LIN {X 0,Y 189.628,Z 761.034,A -85,B 0,C 180,E1 20728.512,E2 20728.512} C_VEL
LIN {X 0,Y 212.096,Z 753.744,A -85,B 0,C 180,E1 20739.808,E2 20739.808} C_VEL
LIN {X 0,Y 217.825,Z 751.684,A -85,B 0,C 180,E1 20741.718,E2 20741.718} C_VEL
LIN {X 0,Y 216.052,Z 752.751,A -85,B 0,C 180,E1 20742.834,E2 20742.834} C_VEL
LIN {X 0,Y 191.697,Z 765.754,A -85,B 0,C 180,E1 20753.818,E2 20753.818} C_VEL
LIN {X 0,Y 179.263,Z 772.931,A -85,B 0,C 180,E1 20765.112,E2 20765.112} C_VEL
LIN {X 0,Y 174.645,Z 775.618,A -85,B 0,C 180,E1 20774.979,E2 20774.979} C_VEL
LIN {X 0,Y 173.679,Z 775.979,A -85,B 0,C 180,E1 20785.018,E2 20785.018} C_VEL
LIN {X 0,Y 173.872,Z 777.551,A -85,B 0,C 180,E1 20790.002,E2 20790.002} C_VEL
LIN {X 0,Y 173.679,Z 777.533,A -85,B 0,C 180,E1 20794.986,E2 20794.986} C_VEL
LIN {X 0,Y 174.385,Z 774.615,A -85,B 0,C 180,E1 20802.496,E2 20802.496} C_VEL
LIN {X 0,Y 177.606,Z 765.224,A -85,B 0,C 180,E1 20812.481,E2 20812.481} C_VEL
LIN {X 0,Y 184.174,Z 750.072,A -85,B 0,C 180,E1 20821.354,E2 20821.354} C_VEL
LIN {X 0,Y 192.922,Z 729.385,A -85,B 0,C 180,E1 20828.739,E2 20828.739} C_VEL
LIN {X 0,Y 201.559,Z 704.57,A -85,B 0,C 180,E1 20834.347,E2 20834.347} C_VEL
LIN {X 0,Y 208.28,Z 677.85,A -85,B 0,C 180,E1 20838.151,E2 20838.151} C_VEL
LIN {X 0,Y 212.35,Z 649.044,A -85,B 0,C 180,E1 20840.62,E2 20840.62} C_VEL
LIN {X 0,Y 213.87,Z 640.631,A -85,B 0,C 180,E1 20841.448,E2 20841.448} C_VEL
LIN {X 0,Y 203.795,Z 603.79,A -85,B 0,C 180,E1 20848.943,E2 20848.943} C_VEL
LIN {X 0,Y 198.917,Z 565.383,A -85,B 0,C 180,E1 20858.768,E2 20858.768} C_VEL
LIN {X 0,Y 197.323,Z 560.632,A -85,B 0,C 180,E1 20863.341,E2 20863.341} C_VEL
LIN {X 0,Y 198.795,Z 561.143,A -85,B 0,C 180,E1 20875.653,E2 20875.653} C_VEL
LIN {X 0,Y 203.113,Z 569.312,A -85,B 0,C 180,E1 20882.168,E2 20882.168} C_VEL
LIN {X 0,Y 209.323,Z 580.62,A -85,B 0,C 180,E1 20887.904,E2 20887.904} C_VEL
LIN {X 0,Y 217.509,Z 597.767,A -85,B 0,C 180,E1 20893.44,E2 20893.44} C_VEL
LIN {X 0,Y 225.175,Z 619.284,A -85,B 0,C 180,E1 20897.758,E2 20897.758} C_VEL
LIN {X 0,Y 226.031,Z 622.404,A -85,B 0,C 180,E1 20898.235,E2 20898.235} C_VEL
LIN {X 0,Y 222.435,Z 652.717,A -85,B 0,C 180,E1 20899.64,E2 20899.64} C_VEL
LIN {X 0,Y 219.352,Z 667.346,A -85,B 0,C 180,E1 20900.828,E2 20900.828} C_VEL
LIN {X 0,Y 212.303,Z 683.08,A -85,B 0,C 180,E1 20901.722,E2 20901.722} C_VEL
LIN {X 0,Y 205.16,Z 696.073,A -85,B 0,C 180,E1 20902.814,E2 20902.814} C_VEL
LIN {X 0,Y 204.418,Z 697.811,A -85,B 0,C 180,E1 20903.1,E2 20903.1} C_VEL
LIN {X 0,Y 194.005,Z 720.009,A -85,B 0,C 180,E1 20907.989,E2 20907.989} C_VEL
LIN {X 0,Y 183.31,Z 738.179,A -85,B 0,C 180,E1 20914.591,E2 20914.591} C_VEL
LIN {X 0,Y 174.062,Z 751.886,A -85,B 0,C 180,E1 20923.249,E2 20923.249} C_VEL
LIN {X 0,Y 169.021,Z 758.609,A -85,B 0,C 180,E1 20931.319,E2 20931.319} C_VEL
LIN {X 0,Y 166.585,Z 760.947,A -85,B 0,C 180,E1 20937.075,E2 20937.075} C_VEL
LIN {X 0,Y 165.326,Z 760.854,A -85,B 0,C 180,E1 20945.902,E2 20945.902} C_VEL
LIN {X 0,Y 167.356,Z 755.765,A -85,B 0,C 180,E1 20955.642,E2 20955.642} C_VEL
LIN {X 0,Y 171.894,Z 745.002,A -85,B 0,C 180,E1 20964.962,E2 20964.962} C_VEL
LIN {X 0,Y 178.888,Z 728.891,A -85,B 0,C 180,E1 20973.02,E2 20973.02} C_VEL
LIN {X 0,Y 187.361,Z 707.541,A -85,B 0,C 180,E1 20979.56,E2 20979.56} C_VEL
LIN {X 0,Y 195.39,Z 682.576,A -85,B 0,C 180,E1 20984.249,E2 20984.249} C_VEL
LIN {X 0,Y 201.6,Z 654.272,A -85,B 0,C 180,E1 20987.42,E2 20987.42} C_VEL
LIN {X 0,Y 205.022,Z 624.843,A -85,B 0,C 180,E1 20989.044,E2 20989.044} C_VEL
LIN {X 0,Y 204.978,Z 613.442,A -85,B 0,C 180,E1 20989.593,E2 20989.593} C_VEL
LIN {X 0,Y 193.143,Z 583.54,A -85,B 0,C 180,E1 20994.123,E2 20994.123} C_VEL
LIN {X 0,Y 184.516,Z 566.701,A -85,B 0,C 180,E1 20997.701,E2 20997.701} C_VEL
LIN {X 0,Y 180.361,Z 568.066,A -85,B 0,C 180,E1 20999.224,E2 20999.224} C_VEL
LIN {X 0,Y 192.479,Z 600.451,A -85,B 0,C 180,E1 21006.012,E2 21006.012} C_VEL
LIN {X 0,Y 201.469,Z 633.152,A -85,B 0,C 180,E1 21012.744,E2 21012.744} C_VEL
LIN {X 0,Y 192.439,Z 663.924,A -85,B 0,C 180,E1 21017.77,E2 21017.77} C_VEL
LIN {X 0,Y 181.952,Z 694.148,A -85,B 0,C 180,E1 21024.976,E2 21024.976} C_VEL
LIN {X 0,Y 173.22,Z 719.714,A -85,B 0,C 180,E1 21034.171,E2 21034.171} C_VEL
LIN {X 0,Y 167.935,Z 738.514,A -85,B 0,C 180,E1 21044.355,E2 21044.355} C_VEL
LIN {X 0,Y 166.031,Z 751.24,A -85,B 0,C 180,E1 21054.779,E2 21054.779} C_VEL
LIN {X 0,Y 166.344,Z 758.967,A -85,B 0,C 180,E1 21065.198,E2 21065.198} C_VEL
LIN {X 0,Y 169.63,Z 762.701,A -85,B 0,C 180,E1 21075.471,E2 21075.471} C_VEL
LIN {X 0,Y 182.8,Z 762.307,A -85,B 0,C 180,E1 21089.681,E2 21089.681} C_VEL
LIN {X 0,Y 207.708,Z 755.77,A -85,B 0,C 180,E1 21101.58,E2 21101.58} C_VEL
LIN {X 0,Y 207.442,Z 756.059,A -85,B 0,C 180,E1 21102.411,E2 21102.411} C_VEL
LIN {X 0,Y 182.073,Z 767.938,A -85,B 0,C 180,E1 21114.541,E2 21114.541} C_VEL
LIN {X 0,Y 168.849,Z 774.269,A -85,B 0,C 180,E1 21129.057,E2 21129.057} C_VEL
LIN {X 0,Y 165.827,Z 774.847,A -85,B 0,C 180,E1 21143.471,E2 21143.471} C_VEL
LIN {X 0,Y 165.967,Z 777.14,A -85,B 0,C 180,E1 21150.134,E2 21150.134} C_VEL
LIN {X 0,Y 165.798,Z 777.161,A -85,B 0,C 180,E1 21155.224,E2 21155.224} C_VEL
LIN {X 0,Y 166.57,Z 774.369,A -85,B 0,C 180,E1 21163.092,E2 21163.092} C_VEL
LIN {X 0,Y 170.156,Z 765.137,A -85,B 0,C 180,E1 21173.523,E2 21173.523} C_VEL
LIN {X 0,Y 177.467,Z 749.999,A -85,B 0,C 180,E1 21182.827,E2 21182.827} C_VEL
LIN {X 0,Y 186.742,Z 729.883,A -85,B 0,C 180,E1 21190.277,E2 21190.277} C_VEL
LIN {X 0,Y 195.714,Z 706.541,A -85,B 0,C 180,E1 21195.771,E2 21195.771} C_VEL
LIN {X 0,Y 203.105,Z 680.501,A -85,B 0,C 180,E1 21199.69,E2 21199.69} C_VEL
LIN {X 0,Y 207.927,Z 651.201,A -85,B 0,C 180,E1 21202.351,E2 21202.351} C_VEL
LIN {X 0,Y 208.329,Z 642.972,A -85,B 0,C 180,E1 21202.993,E2 21202.993} C_VEL
LIN {X 0,Y 198.886,Z 594.701,A -85,B 0,C 180,E1 21213.925,E2 21213.925} C_VEL
LIN {X 0,Y 197.153,Z 572.184,A -85,B 0,C 180,E1 21220.11,E2 21220.11} C_VEL
LIN {X 0,Y 196.152,Z 568.38,A -85,B 0,C 180,E1 21223.777,E2 21223.777} C_VEL
LIN {X 0,Y 197.478,Z 568.897,A -85,B 0,C 180,E1 21235.212,E2 21235.212} C_VEL
LIN {X 0,Y 201.518,Z 576.988,A -85,B 0,C 180,E1 21241.702,E2 21241.702} C_VEL
LIN {X 0,Y 208.238,Z 589.979,A -85,B 0,C 180,E1 21248.076,E2 21248.076} C_VEL
LIN {X 0,Y 216.187,Z 608.855,A -85,B 0,C 180,E1 21253.614,E2 21253.614} C_VEL
LIN {X 0,Y 221.286,Z 624.924,A -85,B 0,C 180,E1 21256.677,E2 21256.677} C_VEL
LIN {X 0,Y 217.341,Z 654.833,A -85,B 0,C 180,E1 21258.13,E2 21258.13} C_VEL
LIN {X 0,Y 209.921,Z 682.887,A -85,B 0,C 180,E1 21260.85,E2 21260.85} C_VEL
LIN {X 0,Y 204.418,Z 697.811,A -85,B 0,C 180,E1 21263.1,E2 21263.1} C_VEL
LIN {X 0,Y 195.677,Z 711.55,A -85,B 0,C 180,E1 21264.989,E2 21264.989} C_VEL
LIN {X 0,Y 187.156,Z 722.49,A -85,B 0,C 180,E1 21266.974,E2 21266.974} C_VEL
LIN {X 0,Y 186.262,Z 723.922,A -85,B 0,C 180,E1 21267.391,E2 21267.391} C_VEL
LIN {X 0,Y 175.216,Z 741.093,A -85,B 0,C 180,E1 21274.304,E2 21274.304} C_VEL
LIN {X 0,Y 165.895,Z 753.645,A -85,B 0,C 180,E1 21283.304,E2 21283.304} C_VEL
LIN {X 0,Y 160.55,Z 759.928,A -85,B 0,C 180,E1 21292.228,E2 21292.228} C_VEL
LIN {X 0,Y 157.683,Z 761.83,A -85,B 0,C 180,E1 21301.411,E2 21301.411} C_VEL
LIN {X 0,Y 158.41,Z 758.563,A -85,B 0,C 180,E1 21312.308,E2 21312.308} C_VEL
LIN {X 0,Y 162.077,Z 750.222,A -85,B 0,C 180,E1 21321.994,E2 21321.994} C_VEL
LIN {X 0,Y 168.815,Z 735.543,A -85,B 0,C 180,E1 21331.278,E2 21331.278} C_VEL
LIN {X 0,Y 177.046,Z 716.518,A -85,B 0,C 180,E1 21338.463,E2 21338.463} C_VEL
LIN {X 0,Y 186.063,Z 692.234,A -85,B 0,C 180,E1 21344.08,E2 21344.08} C_VEL
LIN {X 0,Y 193.442,Z 664.259,A -85,B 0,C 180,E1 21347.933,E2 21347.933} C_VEL
LIN {X 0,Y 198.021,Z 636.087,A -85,B 0,C 180,E1 21350.011,E2 21350.011} C_VEL
LIN {X 0,Y 198.961,Z 616.022,A -85,B 0,C 180,E1 21350.912,E2 21350.912} C_VEL
LIN {X 0,Y 187.164,Z 586.134,A -85,B 0,C 180,E1 21355.733,E2 21355.733} C_VEL
LIN {X 0,Y 181.93,Z 576.305,A -85,B 0,C 180,E1 21357.983,E2 21357.983} C_VEL
LIN {X 0,Y 177.718,Z 578.756,A -85,B 0,C 180,E1 21359.29,E2 21359.29} C_VEL
LIN {X 0,Y 177.042,Z 578.811,A -85,B 0,C 180,E1 21359.673,E2 21359.673} C_VEL
LIN {X 0,Y 187.669,Z 609.878,A -85,B 0,C 180,E1 21366.47,E2 21366.47} C_VEL
LIN {X 0,Y 194.332,Z 635.863,A -85,B 0,C 180,E1 21372.116,E2 21372.116} C_VEL
LIN {X 0,Y 182.885,Z 670.726,A -85,B 0,C 180,E1 21378.229,E2 21378.229} C_VEL
LIN {X 0,Y 172.181,Z 700.201,A -85,B 0,C 180,E1 21386.166,E2 21386.166} C_VEL
LIN {X 0,Y 164.136,Z 723.35,A -85,B 0,C 180,E1 21395.557,E2 21395.557} C_VEL
LIN {X 0,Y 159.49,Z 741.202,A -85,B 0,C 180,E1 21406.311,E2 21406.311} C_VEL
LIN {X 0,Y 157.983,Z 753.046,A -85,B 0,C 180,E1 21417.255,E2 21417.255} C_VEL
LIN {X 0,Y 158.965,Z 760.202,A -85,B 0,C 180,E1 21428.179,E2 21428.179} C_VEL
LIN {X 0,Y 165.439,Z 763.919,A -85,B 0,C 180,E1 21441.39,E2 21441.39} C_VEL
LIN {X 0,Y 183.212,Z 762.391,A -85,B 0,C 180,E1 21455.2,E2 21455.2} C_VEL
LIN {X 0,Y 197.664,Z 759.231,A -85,B 0,C 180,E1 21461.464,E2 21461.464} C_VEL
LIN {X 0,Y 197.434,Z 759.516,A -85,B 0,C 180,E1 21462.426,E2 21462.426} C_VEL
LIN {X 0,Y 172.433,Z 769.611,A -85,B 0,C 180,E1 21475.334,E2 21475.334} C_VEL
LIN {X 0,Y 160.311,Z 774.163,A -85,B 0,C 180,E1 21490.246,E2 21490.246} C_VEL
LIN {X 0,Y 157.942,Z 774.318,A -85,B 0,C 180,E1 21503.143,E2 21503.143} C_VEL
LIN {X 0,Y 158.103,Z 776.683,A -85,B 0,C 180,E1 21510.002,E2 21510.002} C_VEL
LIN {X 0,Y 157.889,Z 776.788,A -85,B 0,C 180,E1 21515.487,E2 21515.487} C_VEL
LIN {X 0,Y 158.753,Z 774.123,A -85,B 0,C 180,E1 21523.749,E2 21523.749} C_VEL
LIN {X 0,Y 162.797,Z 765.073,A -85,B 0,C 180,E1 21534.655,E2 21534.655} C_VEL
LIN {X 0,Y 170.744,Z 750.181,A -85,B 0,C 180,E1 21544.294,E2 21544.294} C_VEL
LIN {X 0,Y 180.725,Z 730.409,A -85,B 0,C 180,E1 21551.914,E2 21551.914} C_VEL
LIN {X 0,Y 190.329,Z 707.567,A -85,B 0,C 180,E1 21557.463,E2 21557.463} C_VEL
LIN {X 0,Y 198.596,Z 680.998,A -85,B 0,C 180,E1 21561.549,E2 21561.549} C_VEL
LIN {X 0,Y 203.976,Z 651.61,A -85,B 0,C 180,E1 21564.25,E2 21564.25} C_VEL
LIN {X 0,Y 204.189,Z 645.575,A -85,B 0,C 180,E1 21564.854,E2 21564.854} C_VEL
LIN {X 0,Y 196.541,Z 598.917,A -85,B 0,C 180,E1 21575.806,E2 21575.806} C_VEL
LIN {X 0,Y 195.582,Z 579.18,A -85,B 0,C 180,E1 21581.253,E2 21581.253} C_VEL
LIN {X 0,Y 194.934,Z 576.15,A -85,B 0,C 180,E1 21584.453,E2 21584.453} C_VEL
LIN {X 0,Y 196.294,Z 576.937,A -85,B 0,C 180,E1 21595.054,E2 21595.054} C_VEL
LIN {X 0,Y 200.005,Z 584.838,A -85,B 0,C 180,E1 21601.317,E2 21601.317} C_VEL
LIN {X 0,Y 205.971,Z 597.331,A -85,B 0,C 180,E1 21607.35,E2 21607.35} C_VEL
LIN {X 0,Y 212.922,Z 614.88,A -85,B 0,C 180,E1 21612.541,E2 21612.541} C_VEL
LIN {X 0,Y 216.636,Z 628.564,A -85,B 0,C 180,E1 21615.096,E2 21615.096} C_VEL
LIN {X 0,Y 212.183,Z 658.001,A -85,B 0,C 180,E1 21616.625,E2 21616.625} C_VEL
LIN {X 0,Y 204.222,Z 685.488,A -85,B 0,C 180,E1 21619.428,E2 21619.428} C_VEL
LIN {X 0,Y 194.017,Z 709.671,A -85,B 0,C 180,E1 21623.652,E2 21623.652} C_VEL
LIN {X 0,Y 186.262,Z 723.922,A -85,B 0,C 180,E1 21627.391,E2 21627.391} C_VEL
LIN {X 0,Y 176.493,Z 734.878,A -85,B 0,C 180,E1 21630.447,E2 21630.447} C_VEL
LIN {X 0,Y 167.686,Z 743.126,A -85,B 0,C 180,E1 21633.613,E2 21633.613} C_VEL
LIN {X 0,Y 166.844,Z 744.164,A -85,B 0,C 180,E1 21634.201,E2 21634.201} C_VEL
LIN {X 0,Y 157.571,Z 755.542,A -85,B 0,C 180,E1 21643.595,E2 21643.595} C_VEL
LIN {X 0,Y 152.001,Z 761.137,A -85,B 0,C 180,E1 21653.438,E2 21653.438} C_VEL
LIN {X 0,Y 150.056,Z 762.194,A -85,B 0,C 180,E1 21659.811,E2 21659.811} C_VEL
LIN {X 0,Y 149.873,Z 760.404,A -85,B 0,C 180,E1 21669.363,E2 21669.363} C_VEL
LIN {X 0,Y 153.178,Z 753.143,A -85,B 0,C 180,E1 21680.145,E2 21680.145} C_VEL
LIN {X 0,Y 159.38,Z 740.172,A -85,B 0,C 180,E1 21689.998,E2 21689.998} C_VEL
LIN {X 0,Y 167.983,Z 721.865,A -85,B 0,C 180,E1 21698.084,E2 21698.084} C_VEL
LIN {X 0,Y 177.152,Z 699.254,A -85,B 0,C 180,E1 21704.173,E2 21704.173} C_VEL
LIN {X 0,Y 185.408,Z 672.3,A -85,B 0,C 180,E1 21708.529,E2 21708.529} C_VEL
LIN {X 0,Y 191.102,Z 643.534,A -85,B 0,C 180,E1 21711.104,E2 21711.104} C_VEL
LIN {X 0,Y 192.851,Z 618.067,A -85,B 0,C 180,E1 21712.373,E2 21712.373} C_VEL
LIN {X 0,Y 181.472,Z 589.025,A -85,B 0,C 180,E1 21717.367,E2 21717.367} C_VEL
LIN {X 0,Y 179.739,Z 586.175,A -85,B 0,C 180,E1 21718.124,E2 21718.124} C_VEL
LIN {X 0,Y 175.253,Z 589.51,A -85,B 0,C 180,E1 21719.489,E2 21719.489} C_VEL
LIN {X 0,Y 173.535,Z 589.694,A -85,B 0,C 180,E1 21720.289,E2 21720.289} C_VEL
LIN {X 0,Y 182.849,Z 620.052,A -85,B 0,C 180,E1 21727.243,E2 21727.243} C_VEL
LIN {X 0,Y 186.67,Z 638.028,A -85,B 0,C 180,E1 21731.303,E2 21731.303} C_VEL
LIN {X 0,Y 174.947,Z 672.291,A -85,B 0,C 180,E1 21737.626,E2 21737.626} C_VEL
LIN {X 0,Y 164.226,Z 701.045,A -85,B 0,C 180,E1 21745.784,E2 21745.784} C_VEL
LIN {X 0,Y 155.999,Z 724.212,A -85,B 0,C 180,E1 21755.718,E2 21755.718} C_VEL
LIN {X 0,Y 151.395,Z 741.872,A -85,B 0,C 180,E1 21767.033,E2 21767.033} C_VEL
LIN {X 0,Y 150.106,Z 753.609,A -85,B 0,C 180,E1 21778.552,E2 21778.552} C_VEL
LIN {X 0,Y 151.972,Z 761.332,A -85,B 0,C 180,E1 21791.447,E2 21791.447} C_VEL
LIN {X 0,Y 163.147,Z 764.871,A -85,B 0,C 180,E1 21807.538,E2 21807.538} C_VEL
LIN {X 0,Y 188.299,Z 761.982,A -85,B 0,C 180,E1 21821.617,E2 21821.617} C_VEL
LIN {X 0,Y 176.931,Z 765.985,A -85,B 0,C 180,E1 21826.98,E2 21826.98} C_VEL
LIN {X 0,Y 157.636,Z 772.371,A -85,B 0,C 180,E1 21841.407,E2 21841.407} C_VEL
LIN {X 0,Y 150.423,Z 773.203,A -85,B 0,C 180,E1 21858.429,E2 21858.429} C_VEL
LIN {X 0,Y 150.174,Z 772.989,A -85,B 0,C 180,E1 21861.334,E2 21861.334} C_VEL
LIN {X 0,Y 150.225,Z 776.245,A -85,B 0,C 180,E1 21870.002,E2 21870.002} C_VEL
LIN {X 0,Y 149.986,Z 776.416,A -85,B 0,C 180,E1 21875.777,E2 21875.777} C_VEL
LIN {X 0,Y 150.972,Z 773.862,A -85,B 0,C 180,E1 21884.473,E2 21884.473} C_VEL
LIN {X 0,Y 155.506,Z 765.02,A -85,B 0,C 180,E1 21895.894,E2 21895.894} C_VEL
LIN {X 0,Y 164.155,Z 750.364,A -85,B 0,C 180,E1 21905.878,E2 21905.878} C_VEL
LIN {X 0,Y 174.871,Z 731.01,A -85,B 0,C 180,E1 21913.66,E2 21913.66} C_VEL
LIN {X 0,Y 185.907,Z 706.743,A -85,B 0,C 180,E1 21919.615,E2 21919.615} C_VEL
LIN {X 0,Y 194.859,Z 679.634,A -85,B 0,C 180,E1 21923.714,E2 21923.714} C_VEL
LIN {X 0,Y 200.409,Z 649.217,A -85,B 0,C 180,E1 21926.563,E2 21926.563} C_VEL
LIN {X 0,Y 194.426,Z 602.064,A -85,B 0,C 180,E1 21937.983,E2 21937.983} C_VEL
LIN {X 0,Y 194.16,Z 586.04,A -85,B 0,C 180,E1 21942.507,E2 21942.507} C_VEL
LIN {X 0,Y 193.742,Z 583.92,A -85,B 0,C 180,E1 21945.136,E2 21945.136} C_VEL
LIN {X 0,Y 195.011,Z 584.643,A -85,B 0,C 180,E1 21954.595,E2 21954.595} C_VEL
LIN {X 0,Y 198.777,Z 593.064,A -85,B 0,C 180,E1 21961.236,E2 21961.236} C_VEL
LIN {X 0,Y 204.715,Z 606.886,A -85,B 0,C 180,E1 21967.435,E2 21967.435} C_VEL
LIN {X 0,Y 211.136,Z 625.779,A -85,B 0,C 180,E1 21972.483,E2 21972.483} C_VEL
LIN {X 0,Y 212.219,Z 630.971,A -85,B 0,C 180,E1 21973.385,E2 21973.385} C_VEL
LIN {X 0,Y 207.312,Z 660.175,A -85,B 0,C 180,E1 21974.974,E2 21974.974} C_VEL
LIN {X 0,Y 198.833,Z 687.616,A -85,B 0,C 180,E1 21977.863,E2 21977.863} C_VEL
LIN {X 0,Y 187.723,Z 712.088,A -85,B 0,C 180,E1 21982.312,E2 21982.312} C_VEL
LIN {X 0,Y 175.442,Z 732.306,A -85,B 0,C 180,E1 21988.436,E2 21988.436} C_VEL
LIN {X 0,Y 166.844,Z 744.164,A -85,B 0,C 180,E1 21994.201,E2 21994.201} C_VEL
LIN {X 0,Y 157.636,Z 751.717,A -85,B 0,C 180,E1 21998.746,E2 21998.746} C_VEL
LIN {X 0,Y 149.113,Z 757.363,A -85,B 0,C 180,E1 22004.075,E2 22004.075} C_VEL
LIN {X 0,Y 144.969,Z 761.155,A -85,B 0,C 180,E1 22011.348,E2 22011.348} C_VEL
LIN {X 0,Y 142.516,Z 762.55,A -85,B 0,C 180,E1 22018.031,E2 22018.031} C_VEL
LIN {X 0,Y 141.776,Z 761.214,A -85,B 0,C 180,E1 22028.126,E2 22028.126} C_VEL
LIN {X 0,Y 145.085,Z 754.21,A -85,B 0,C 180,E1 22039.906,E2 22039.906} C_VEL
LIN {X 0,Y 151.179,Z 742.096,A -85,B 0,C 180,E1 22049.998,E2 22049.998} C_VEL
LIN {X 0,Y 159.434,Z 725.534,A -85,B 0,C 180,E1 22058.158,E2 22058.158} C_VEL
LIN {X 0,Y 169.28,Z 703.118,A -85,B 0,C 180,E1 22064.847,E2 22064.847} C_VEL
LIN {X 0,Y 178.381,Z 676.175,A -85,B 0,C 180,E1 22069.598,E2 22069.598} C_VEL
LIN {X 0,Y 184.523,Z 647.904,A -85,B 0,C 180,E1 22072.416,E2 22072.416} C_VEL
LIN {X 0,Y 187.067,Z 620.816,A -85,B 0,C 180,E1 22073.825,E2 22073.825} C_VEL
LIN {X 0,Y 177.841,Z 596.291,A -85,B 0,C 180,E1 22078.147,E2 22078.147} C_VEL
LIN {X 0,Y 170.407,Z 600.502,A -85,B 0,C 180,E1 22080.569,E2 22080.569} C_VEL
LIN {X 0,Y 169.696,Z 600.579,A -85,B 0,C 180,E1 22081.052,E2 22081.052} C_VEL
LIN {X 0,Y 178.051,Z 631.757,A -85,B 0,C 180,E1 22088.546,E2 22088.546} C_VEL
LIN {X 0,Y 179.24,Z 639.536,A -85,B 0,C 180,E1 22090.354,E2 22090.354} C_VEL
LIN {X 0,Y 167.255,Z 673.247,A -85,B 0,C 180,E1 22096.86,E2 22096.86} C_VEL
LIN {X 0,Y 156.233,Z 701.911,A -85,B 0,C 180,E1 22105.419,E2 22105.419} C_VEL
LIN {X 0,Y 147.833,Z 724.983,A -85,B 0,C 180,E1 22115.894,E2 22115.894} C_VEL
LIN {X 0,Y 143.328,Z 742.475,A -85,B 0,C 180,E1 22127.836,E2 22127.836} C_VEL
LIN {X 0,Y 142.307,Z 754.116,A -85,B 0,C 180,E1 22139.992,E2 22139.992} C_VEL
LIN {X 0,Y 144.21,Z 761.258,A -85,B 0,C 180,E1 22152.072,E2 22152.072} C_VEL
LIN {X 0,Y 156.198,Z 765.58,A -85,B 0,C 180,E1 22168.875,E2 22168.875} C_VEL
LIN {X 0,Y 178.13,Z 764.364,A -85,B 0,C 180,E1 22181.495,E2 22181.495} C_VEL
LIN {X 0,Y 176.293,Z 765.001,A -85,B 0,C 180,E1 22182.838,E2 22182.838} C_VEL
LIN {X 0,Y 150.624,Z 771.993,A -85,B 0,C 180,E1 22199.942,E2 22199.942} C_VEL
LIN {X 0,Y 142.646,Z 772.227,A -85,B 0,C 180,E1 22217.788,E2 22217.788} C_VEL
LIN {X 0,Y 142.349,Z 772.425,A -85,B 0,C 180,E1 22220.853,E2 22220.853} C_VEL
LIN {X 0,Y 142.32,Z 775.803,A -85,B 0,C 180,E1 22230.003,E2 22230.003} C_VEL
LIN {X 0,Y 142.078,Z 776.044,A -85,B 0,C 180,E1 22236.099,E2 22236.099} C_VEL
LIN {X 0,Y 143.207,Z 773.601,A -85,B 0,C 180,E1 22245.276,E2 22245.276} C_VEL
LIN {X 0,Y 148.304,Z 764.995,A -85,B 0,C 180,E1 22257.253,E2 22257.253} C_VEL
LIN {X 0,Y 157.692,Z 750.587,A -85,B 0,C 180,E1 22267.595,E2 22267.595} C_VEL
LIN {X 0,Y 169.211,Z 731.612,A -85,B 0,C 180,E1 22275.517,E2 22275.517} C_VEL
LIN {X 0,Y 180.478,Z 708.981,A -85,B 0,C 180,E1 22281.286,E2 22281.286} C_VEL
LIN {X 0,Y 189.959,Z 683.295,A -85,B 0,C 180,E1 22285.385,E2 22285.385} C_VEL
LIN {X 0,Y 196.796,Z 652.858,A -85,B 0,C 180,E1 22288.331,E2 22288.331} C_VEL
LIN {X 0,Y 192.592,Z 604.507,A -85,B 0,C 180,E1 22300.384,E2 22300.384} C_VEL
LIN {X 0,Y 192.834,Z 592.695,A -85,B 0,C 180,E1 22303.915,E2 22303.915} C_VEL
LIN {X 0,Y 192.853,Z 591.48,A -85,B 0,C 180,E1 22311.003,E2 22311.003} C_VEL
LIN {X 0,Y 193.939,Z 592.919,A -85,B 0,C 180,E1 22314.705,E2 22314.705} C_VEL
LIN {X 0,Y 197.491,Z 601.298,A -85,B 0,C 180,E1 22321.089,E2 22321.089} C_VEL
LIN {X 0,Y 203.135,Z 615.947,A -85,B 0,C 180,E1 22327.259,E2 22327.259} C_VEL
LIN {X 0,Y 208.085,Z 632.68,A -85,B 0,C 180,E1 22331.523,E2 22331.523} C_VEL
LIN {X 0,Y 202.816,Z 662.049,A -85,B 0,C 180,E1 22333.209,E2 22333.209} C_VEL
LIN {X 0,Y 193.83,Z 689.253,A -85,B 0,C 180,E1 22336.144,E2 22336.144} C_VEL
LIN {X 0,Y 181.769,Z 714.063,A -85,B 0,C 180,E1 22340.802,E2 22340.802} C_VEL
LIN {X 0,Y 169.187,Z 733.463,A -85,B 0,C 180,E1 22346.882,E2 22346.882} C_VEL
LIN {X 0,Y 157.189,Z 748.569,A -85,B 0,C 180,E1 22355.178,E2 22355.178} C_VEL
LIN {X 0,Y 149.113,Z 757.363,A -85,B 0,C 180,E1 22364.075,E2 22364.075} C_VEL
LIN {X 0,Y 143.739,Z 760.436,A -85,B 0,C 180,E1 22368.613,E2 22368.613} C_VEL
LIN {X 0,Y 135.213,Z 762.818,A -85,B 0,C 180,E1 22375.929,E2 22375.929} C_VEL
LIN {X 0,Y 134.834,Z 762.825,A -85,B 0,C 180,E1 22376.85,E2 22376.85} C_VEL
LIN {X 0,Y 133.728,Z 762.462,A -85,B 0,C 180,E1 22384.537,E2 22384.537} C_VEL
LIN {X 0,Y 136.034,Z 757.056,A -85,B 0,C 180,E1 22397.179,E2 22397.179} C_VEL
LIN {X 0,Y 141.786,Z 746.054,A -85,B 0,C 180,E1 22408.473,E2 22408.473} C_VEL
LIN {X 0,Y 150.438,Z 729.936,A -85,B 0,C 180,E1 22417.8,E2 22417.8} C_VEL
LIN {X 0,Y 160.484,Z 709.031,A -85,B 0,C 180,E1 22424.983,E2 22424.983} C_VEL
LIN {X 0,Y 170.049,Z 683.806,A -85,B 0,C 180,E1 22430.157,E2 22430.157} C_VEL
LIN {X 0,Y 177.316,Z 655.689,A -85,B 0,C 180,E1 22433.502,E2 22433.502} C_VEL
LIN {X 0,Y 181.379,Z 625.224,A -85,B 0,C 180,E1 22435.256,E2 22435.256} C_VEL
LIN {X 0,Y 175.984,Z 607.958,A -85,B 0,C 180,E1 22438.058,E2 22438.058} C_VEL
LIN {X 0,Y 170.976,Z 608.808,A -85,B 0,C 180,E1 22439.793,E2 22439.793} C_VEL
LIN {X 0,Y 167.395,Z 611.489,A -85,B 0,C 180,E1 22440.985,E2 22440.985} C_VEL
LIN {X 0,Y 165.424,Z 611.345,A -85,B 0,C 180,E1 22441.922,E2 22441.922} C_VEL
LIN {X 0,Y 172.131,Z 640.155,A -85,B 0,C 180,E1 22449.214,E2 22449.214} C_VEL
LIN {X 0,Y 159.427,Z 674.544,A -85,B 0,C 180,E1 22456.147,E2 22456.147} C_VEL
LIN {X 0,Y 148.134,Z 702.785,A -85,B 0,C 180,E1 22465.055,E2 22465.055} C_VEL
LIN {X 0,Y 139.363,Z 726.814,A -85,B 0,C 180,E1 22476.765,E2 22476.765} C_VEL
LIN {X 0,Y 135.1,Z 744.15,A -85,B 0,C 180,E1 22489.802,E2 22489.802} C_VEL
LIN {X 0,Y 134.573,Z 755.654,A -85,B 0,C 180,E1 22503.205,E2 22503.205} C_VEL
LIN {X 0,Y 139.305,Z 763.478,A -85,B 0,C 180,E1 22518.955,E2 22518.955} C_VEL
LIN {X 0,Y 156.335,Z 766.521,A -85,B 0,C 180,E1 22535.38,E2 22535.38} C_VEL
LIN {X 0,Y 167.045,Z 766.219,A -85,B 0,C 180,E1 22540.963,E2 22540.963} C_VEL
LIN {X 0,Y 167.99,Z 766.334,A -85,B 0,C 180,E1 22542.149,E2 22542.149} C_VEL
LIN {X 0,Y 143.704,Z 771.569,A -85,B 0,C 180,E1 22558.333,E2 22558.333} C_VEL
LIN {X 0,Y 134.828,Z 770.937,A -85,B 0,C 180,E1 22577.889,E2 22577.889} C_VEL
LIN {X 0,Y 134.421,Z 775.359,A -85,B 0,C 180,E1 22590.003,E2 22590.003} C_VEL
LIN {X 0,Y 134.178,Z 775.674,A -85,B 0,C 180,E1 22596.46,E2 22596.46} C_VEL
LIN {X 0,Y 135.492,Z 773.351,A -85,B 0,C 180,E1 22606.169,E2 22606.169} C_VEL
LIN {X 0,Y 141.208,Z 764.976,A -85,B 0,C 180,E1 22618.746,E2 22618.746} C_VEL
LIN {X 0,Y 151.396,Z 750.83,A -85,B 0,C 180,E1 22629.453,E2 22629.453} C_VEL
LIN {X 0,Y 163.734,Z 732.201,A -85,B 0,C 180,E1 22637.504,E2 22637.504} C_VEL
LIN {X 0,Y 176.392,Z 708.649,A -85,B 0,C 180,E1 22643.593,E2 22643.593} C_VEL
LIN {X 0,Y 187.2,Z 680.965,A -85,B 0,C 180,E1 22647.857,E2 22647.857} C_VEL
LIN {X 0,Y 193.234,Z 655.109,A -85,B 0,C 180,E1 22650.483,E2 22650.483} C_VEL
LIN {X 0,Y 191.241,Z 606.707,A -85,B 0,C 180,E1 22662.883,E2 22662.883} C_VEL
LIN {X 0,Y 191.645,Z 599.728,A -85,B 0,C 180,E1 22664.97,E2 22664.97} C_VEL
LIN {X 0,Y 192.618,Z 600.296,A -85,B 0,C 180,E1 22673.963,E2 22673.963} C_VEL
LIN {X 0,Y 195.759,Z 608.661,A -85,B 0,C 180,E1 22680.318,E2 22680.318} C_VEL
LIN {X 0,Y 200.726,Z 622.797,A -85,B 0,C 180,E1 22686.281,E2 22686.281} C_VEL
LIN {X 0,Y 204.066,Z 635.421,A -85,B 0,C 180,E1 22689.641,E2 22689.641} C_VEL
LIN {X 0,Y 198.306,Z 664.935,A -85,B 0,C 180,E1 22691.453,E2 22691.453} C_VEL
LIN {X 0,Y 189.099,Z 690.799,A -85,B 0,C 180,E1 22694.31,E2 22694.31} C_VEL
LIN {X 0,Y 176.703,Z 714.869,A -85,B 0,C 180,E1 22698.885,E2 22698.885} C_VEL
LIN {X 0,Y 163.048,Z 734.642,A -85,B 0,C 180,E1 22705.224,E2 22705.224} C_VEL
LIN {X 0,Y 150.142,Z 749.671,A -85,B 0,C 180,E1 22713.911,E2 22713.911} C_VEL
LIN {X 0,Y 141.636,Z 758.173,A -85,B 0,C 180,E1 22723.149,E2 22723.149} C_VEL
LIN {X 0,Y 137.507,Z 761.555,A -85,B 0,C 180,E1 22730.202,E2 22730.202} C_VEL
LIN {X 0,Y 134.834,Z 762.825,A -85,B 0,C 180,E1 22736.85,E2 22736.85} C_VEL
LIN {X 0,Y 131.272,Z 762.945,A -85,B 0,C 180,E1 22742.267,E2 22742.267} C_VEL
LIN {X 0,Y 126.408,Z 760.942,A -85,B 0,C 180,E1 22750.734,E2 22750.734} C_VEL
LIN {X 0,Y 126.512,Z 760.503,A -85,B 0,C 180,E1 22751.71,E2 22751.71} C_VEL
LIN {X 0,Y 130.608,Z 752.963,A -85,B 0,C 180,E1 22763.363,E2 22763.363} C_VEL
LIN {X 0,Y 137.849,Z 740.17,A -85,B 0,C 180,E1 22773.913,E2 22773.913} C_VEL
LIN {X 0,Y 147.652,Z 722.244,A -85,B 0,C 180,E1 22782.541,E2 22782.541} C_VEL
LIN {X 0,Y 158.113,Z 699.718,A -85,B 0,C 180,E1 22789.002,E2 22789.002} C_VEL
LIN {X 0,Y 167.219,Z 673.488,A -85,B 0,C 180,E1 22793.427,E2 22793.427} C_VEL
LIN {X 0,Y 173.767,Z 643.678,A -85,B 0,C 180,E1 22796.177,E2 22796.177} C_VEL
LIN {X 0,Y 175.287,Z 624.521,A -85,B 0,C 180,E1 22797.262,E2 22797.262} C_VEL
LIN {X 0,Y 171.988,Z 616.681,A -85,B 0,C 180,E1 22798.902,E2 22798.902} C_VEL
LIN {X 0,Y 165.499,Z 621.186,A -85,B 0,C 180,E1 22801.05,E2 22801.05} C_VEL
LIN {X 0,Y 161.343,Z 622.854,A -85,B 0,C 180,E1 22802.663,E2 22802.663} C_VEL
LIN {X 0,Y 160.815,Z 623.153,A -85,B 0,C 180,E1 22803.197,E2 22803.197} C_VEL
LIN {X 0,Y 164.733,Z 641.513,A -85,B 0,C 180,E1 22808.123,E2 22808.123} C_VEL
LIN {X 0,Y 151.77,Z 675.317,A -85,B 0,C 180,E1 22815.257,E2 22815.257} C_VEL
LIN {X 0,Y 140.128,Z 703.503,A -85,B 0,C 180,E1 22824.637,E2 22824.637} C_VEL
LIN {X 0,Y 131.302,Z 727.081,A -85,B 0,C 180,E1 22836.831,E2 22836.831} C_VEL
LIN {X 0,Y 127.242,Z 743.46,A -85,B 0,C 180,E1 22849.744,E2 22849.744} C_VEL
LIN {X 0,Y 126.72,Z 754.936,A -85,B 0,C 180,E1 22863.404,E2 22863.404} C_VEL
LIN {X 0,Y 131.828,Z 763.337,A -85,B 0,C 180,E1 22880.075,E2 22880.075} C_VEL
LIN {X 0,Y 149.997,Z 767.313,A -85,B 0,C 180,E1 22897.119,E2 22897.119} C_VEL
LIN {X 0,Y 158.747,Z 767.442,A -85,B 0,C 180,E1 22901.702,E2 22901.702} C_VEL
LIN {X 0,Y 136.923,Z 770.961,A -85,B 0,C 180,E1 22916.565,E2 22916.565} C_VEL
LIN {X 0,Y 126.96,Z 770.252,A -85,B 0,C 180,E1 22937.998,E2 22937.998} C_VEL
LIN {X 0,Y 126.515,Z 774.912,A -85,B 0,C 180,E1 22950.003,E2 22950.003} C_VEL
LIN {X 0,Y 126.274,Z 775.304,A -85,B 0,C 180,E1 22956.866,E2 22956.866} C_VEL
LIN {X 0,Y 127.779,Z 773.148,A -85,B 0,C 180,E1 22967.059,E2 22967.059} C_VEL
LIN {X 0,Y 134.189,Z 764.938,A -85,B 0,C 180,E1 22980.403,E2 22980.403} C_VEL
LIN {X 0,Y 145.281,Z 751.115,A -85,B 0,C 180,E1 22991.468,E2 22991.468} C_VEL
LIN {X 0,Y 158.477,Z 732.855,A -85,B 0,C 180,E1 22999.622,E2 22999.622} C_VEL
LIN {X 0,Y 172.024,Z 709.643,A -85,B 0,C 180,E1 23005.745,E2 23005.745} C_VEL
LIN {X 0,Y 183.244,Z 683.389,A -85,B 0,C 180,E1 23009.854,E2 23009.854} C_VEL
LIN {X 0,Y 189.928,Z 658.337,A -85,B 0,C 180,E1 23012.488,E2 23012.488} C_VEL
LIN {X 0,Y 189.525,Z 621.676,A -85,B 0,C 180,E1 23021.986,E2 23021.986} C_VEL
LIN {X 0,Y 190.428,Z 607.245,A -85,B 0,C 180,E1 23026.254,E2 23026.254} C_VEL
LIN {X 0,Y 191.424,Z 608.167,A -85,B 0,C 180,E1 23033.642,E2 23033.642} C_VEL
LIN {X 0,Y 194.269,Z 616.576,A -85,B 0,C 180,E1 23039.867,E2 23039.867} C_VEL
LIN {X 0,Y 198.665,Z 630.694,A -85,B 0,C 180,E1 23045.613,E2 23045.613} C_VEL
LIN {X 0,Y 200.271,Z 639.606,A -85,B 0,C 180,E1 23047.855,E2 23047.855} C_VEL
LIN {X 0,Y 193.916,Z 667.701,A -85,B 0,C 180,E1 23049.612,E2 23049.612} C_VEL
LIN {X 0,Y 183.608,Z 694.381,A -85,B 0,C 180,E1 23052.682,E2 23052.682} C_VEL
LIN {X 0,Y 171.189,Z 716.808,A -85,B 0,C 180,E1 23057.112,E2 23057.112} C_VEL
LIN {X 0,Y 157.355,Z 735.511,A -85,B 0,C 180,E1 23063.287,E2 23063.287} C_VEL
LIN {X 0,Y 143.175,Z 750.773,A -85,B 0,C 180,E1 23072.52,E2 23072.52} C_VEL
LIN {X 0,Y 133.871,Z 759.189,A -85,B 0,C 180,E1 23082.568,E2 23082.568} C_VEL
LIN {X 0,Y 127.019,Z 763.34,A -85,B 0,C 180,E1 23096.402,E2 23096.402} C_VEL
LIN {X 0,Y 126.068,Z 761.599,A -85,B 0,C 180,E1 23108.953,E2 23108.953} C_VEL
LIN {X 0,Y 126.512,Z 760.503,A -85,B 0,C 180,E1 23111.71,E2 23111.71} C_VEL
LIN {X 0,Y 125.588,Z 757.701,A -85,B 0,C 180,E1 23117.537,E2 23117.537} C_VEL
LIN {X 0,Y 124.125,Z 751.424,A -85,B 0,C 180,E1 23126.206,E2 23126.206} C_VEL
LIN {X 0,Y 124.574,Z 750.527,A -85,B 0,C 180,E1 23127.114,E2 23127.114} C_VEL
LIN {X 0,Y 133.55,Z 735.687,A -85,B 0,C 180,E1 23138.117,E2 23138.117} C_VEL
LIN {X 0,Y 143.901,Z 716.939,A -85,B 0,C 180,E1 23146.188,E2 23146.188} C_VEL
LIN {X 0,Y 154.715,Z 693.356,A -85,B 0,C 180,E1 23152.159,E2 23152.159} C_VEL
LIN {X 0,Y 163.486,Z 666.193,A -85,B 0,C 180,E1 23156.185,E2 23156.185} C_VEL
LIN {X 0,Y 169.148,Z 637.18,A -85,B 0,C 180,E1 23158.431,E2 23158.431} C_VEL
LIN {X 0,Y 169.755,Z 626.97,A -85,B 0,C 180,E1 23159.025,E2 23159.025} C_VEL
LIN {X 0,Y 168.228,Z 627.206,A -85,B 0,C 180,E1 23159.572,E2 23159.572} C_VEL
LIN {X 0,Y 157.403,Z 634.216,A -85,B 0,C 180,E1 23163.476,E2 23163.476} C_VEL
LIN {X 0,Y 155.757,Z 634.079,A -85,B 0,C 180,E1 23164.474,E2 23164.474} C_VEL
LIN {X 0,Y 157.119,Z 643.607,A -85,B 0,C 180,E1 23167.104,E2 23167.104} C_VEL
LIN {X 0,Y 143.938,Z 676.455,A -85,B 0,C 180,E1 23174.412,E2 23174.412} C_VEL
LIN {X 0,Y 132.163,Z 703.969,A -85,B 0,C 180,E1 23184.103,E2 23184.103} C_VEL
LIN {X 0,Y 123.251,Z 727.151,A -85,B 0,C 180,E1 23196.84,E2 23196.84} C_VEL
LIN {X 0,Y 119.188,Z 743.828,A -85,B 0,C 180,E1 23210.885,E2 23210.885} C_VEL
LIN {X 0,Y 119.059,Z 755.252,A -85,B 0,C 180,E1 23225.445,E2 23225.445} C_VEL
LIN {X 0,Y 124.435,Z 763.152,A -85,B 0,C 180,E1 23241.324,E2 23241.324} C_VEL
LIN {X 0,Y 146.597,Z 768.074,A -85,B 0,C 180,E1 23260.56,E2 23260.56} C_VEL
LIN {X 0,Y 147.865,Z 768.163,A -85,B 0,C 180,E1 23261.215,E2 23261.215} C_VEL
LIN {X 0,Y 145.539,Z 768.661,A -85,B 0,C 180,E1 23263.47,E2 23263.47} C_VEL
LIN {X 0,Y 124.994,Z 770.332,A -85,B 0,C 180,E1 23281.128,E2 23281.128} C_VEL
LIN {X 0,Y 119.36,Z 769.078,A -85,B 0,C 180,E1 23296.291,E2 23296.291} C_VEL
LIN {X 0,Y 118.635,Z 774.446,A -85,B 0,C 180,E1 23310.003,E2 23310.003} C_VEL
LIN {X 0,Y 118.404,Z 774.937,A -85,B 0,C 180,E1 23317.325,E2 23317.325} C_VEL
LIN {X 0,Y 120.039,Z 773.025,A -85,B 0,C 180,E1 23327.868,E2 23327.868} C_VEL
LIN {X 0,Y 127.289,Z 764.917,A -85,B 0,C 180,E1 23342.243,E2 23342.243} C_VEL
LIN {X 0,Y 139.374,Z 751.427,A -85,B 0,C 180,E1 23353.651,E2 23353.651} C_VEL
LIN {X 0,Y 154.631,Z 731.876,A -85,B 0,C 180,E1 23362.461,E2 23362.461} C_VEL
LIN {X 0,Y 168.553,Z 709.443,A -85,B 0,C 180,E1 23368.265,E2 23368.265} C_VEL
LIN {X 0,Y 180.331,Z 683.478,A -85,B 0,C 180,E1 23372.215,E2 23372.215} C_VEL
LIN {X 0,Y 186.817,Z 661.136,A -85,B 0,C 180,E1 23374.645,E2 23374.645} C_VEL
LIN {X 0,Y 188.269,Z 626.82,A -85,B 0,C 180,E1 23383.762,E2 23383.762} C_VEL
LIN {X 0,Y 189.295,Z 615.048,A -85,B 0,C 180,E1 23387.133,E2 23387.133} C_VEL
LIN {X 0,Y 190.223,Z 615.965,A -85,B 0,C 180,E1 23393.251,E2 23393.251} C_VEL
LIN {X 0,Y 192.737,Z 624.276,A -85,B 0,C 180,E1 23399.305,E2 23399.305} C_VEL
LIN {X 0,Y 196.14,Z 637.597,A -85,B 0,C 180,E1 23404.572,E2 23404.572} C_VEL
LIN {X 0,Y 196.704,Z 642.928,A -85,B 0,C 180,E1 23405.879,E2 23405.879} C_VEL
LIN {X 0,Y 189.29,Z 672.228,A -85,B 0,C 180,E1 23407.845,E2 23407.845} C_VEL
LIN {X 0,Y 178.287,Z 697.829,A -85,B 0,C 180,E1 23410.953,E2 23410.953} C_VEL
LIN {X 0,Y 164.771,Z 720.133,A -85,B 0,C 180,E1 23415.601,E2 23415.601} C_VEL
LIN {X 0,Y 149.719,Z 738.758,A -85,B 0,C 180,E1 23422.296,E2 23422.296} C_VEL
LIN {X 0,Y 136.646,Z 751.624,A -85,B 0,C 180,E1 23430.736,E2 23430.736} C_VEL
LIN {X 0,Y 126.363,Z 760.009,A -85,B 0,C 180,E1 23441.548,E2 23441.548} C_VEL
LIN {X 0,Y 120.816,Z 763.305,A -85,B 0,C 180,E1 23451.351,E2 23451.351} C_VEL
LIN {X 0,Y 117.946,Z 763.241,A -85,B 0,C 180,E1 23463.603,E2 23463.603} C_VEL
LIN {X 0,Y 120.07,Z 758.25,A -85,B 0,C 180,E1 23477.157,E2 23477.157} C_VEL
LIN {X 0,Y 124.574,Z 750.527,A -85,B 0,C 180,E1 23487.114,E2 23487.114} C_VEL
LIN {X 0,Y 125.718,Z 744.971,A -85,B 0,C 180,E1 23492.517,E2 23492.517} C_VEL
LIN {X 0,Y 127.263,Z 735.007,A -85,B 0,C 180,E1 23500.275,E2 23500.275} C_VEL
LIN {X 0,Y 127.992,Z 733.711,A -85,B 0,C 180,E1 23501.011,E2 23501.011} C_VEL
LIN {X 0,Y 139.691,Z 713.208,A -85,B 0,C 180,E1 23509.316,E2 23509.316} C_VEL
LIN {X 0,Y 150.827,Z 688.49,A -85,B 0,C 180,E1 23515.093,E2 23515.093} C_VEL
LIN {X 0,Y 159.541,Z 660.242,A -85,B 0,C 180,E1 23518.805,E2 23518.805} C_VEL
LIN {X 0,Y 163.668,Z 638.4,A -85,B 0,C 180,E1 23520.375,E2 23520.375} C_VEL
LIN {X 0,Y 152.262,Z 644.807,A -85,B 0,C 180,E1 23524.616,E2 23524.616} C_VEL
LIN {X 0,Y 149.738,Z 645.028,A -85,B 0,C 180,E1 23525.89,E2 23525.89} C_VEL
LIN {X 0,Y 135.776,Z 678.334,A -85,B 0,C 180,E1 23533.736,E2 23533.736} C_VEL
LIN {X 0,Y 123.344,Z 706.325,A -85,B 0,C 180,E1 23544.46,E2 23544.46} C_VEL
LIN {X 0,Y 114.388,Z 729.587,A -85,B 0,C 180,E1 23558.719,E2 23558.719} C_VEL
LIN {X 0,Y 111.214,Z 744.125,A -85,B 0,C 180,E1 23572.191,E2 23572.191} C_VEL
LIN {X 0,Y 111.604,Z 755.503,A -85,B 0,C 180,E1 23587.76,E2 23587.76} C_VEL
LIN {X 0,Y 119.566,Z 764.097,A -85,B 0,C 180,E1 23606.203,E2 23606.203} C_VEL
LIN {X 0,Y 137.742,Z 768.343,A -85,B 0,C 180,E1 23621.083,E2 23621.083} C_VEL
LIN {X 0,Y 131.284,Z 769.105,A -85,B 0,C 180,E1 23626.402,E2 23626.402} C_VEL
LIN {X 0,Y 113.293,Z 768.17,A -85,B 0,C 180,E1 23648.775,E2 23648.775} C_VEL
LIN {X 0,Y 111.852,Z 767.778,A -85,B 0,C 180,E1 23654.35,E2 23654.35} C_VEL
LIN {X 0,Y 110.487,Z 773.019,A -85,B 0,C 180,E1 23666.088,E2 23666.088} C_VEL
LIN {X 0,Y 110.728,Z 773.948,A -85,B 0,C 180,E1 23670.003,E2 23670.003} C_VEL
LIN {X 0,Y 110.51,Z 774.552,A -85,B 0,C 180,E1 23677.852,E2 23677.852} C_VEL
LIN {X 0,Y 112.858,Z 772.284,A -85,B 0,C 180,E1 23690.649,E2 23690.649} C_VEL
LIN {X 0,Y 120.553,Z 764.907,A -85,B 0,C 180,E1 23704.286,E2 23704.286} C_VEL
LIN {X 0,Y 133.705,Z 751.709,A -85,B 0,C 180,E1 23716.016,E2 23716.016} C_VEL
LIN {X 0,Y 149.811,Z 732.844,A -85,B 0,C 180,E1 23724.787,E2 23724.787} C_VEL
LIN {X 0,Y 165.297,Z 709.506,A -85,B 0,C 180,E1 23730.809,E2 23730.809} C_VEL
LIN {X 0,Y 177.988,Z 683.102,A -85,B 0,C 180,E1 23734.726,E2 23734.726} C_VEL
LIN {X 0,Y 183.956,Z 664.701,A -85,B 0,C 180,E1 23736.703,E2 23736.703} C_VEL
LIN {X 0,Y 187.308,Z 630.759,A -85,B 0,C 180,E1 23745.904,E2 23745.904} C_VEL
LIN {X 0,Y 188.211,Z 622.847,A -85,B 0,C 180,E1 23748.195,E2 23748.195} C_VEL
LIN {X 0,Y 189.053,Z 623.843,A -85,B 0,C 180,E1 23752.955,E2 23752.955} C_VEL
LIN {X 0,Y 191.348,Z 632.596,A -85,B 0,C 180,E1 23759.018,E2 23759.018} C_VEL
LIN {X 0,Y 193.569,Z 645.133,A -85,B 0,C 180,E1 23763.777,E2 23763.777} C_VEL
LIN {X 0,Y 185.88,Z 673.628,A -85,B 0,C 180,E1 23765.713,E2 23765.713} C_VEL
LIN {X 0,Y 173.639,Z 700.423,A -85,B 0,C 180,E1 23768.976,E2 23768.976} C_VEL
LIN {X 0,Y 158.315,Z 723.627,A -85,B 0,C 180,E1 23774.033,E2 23774.033} C_VEL
LIN {X 0,Y 141.863,Z 742.071,A -85,B 0,C 180,E1 23781.351,E2 23781.351} C_VEL
LIN {X 0,Y 126.962,Z 755.089,A -85,B 0,C 180,E1 23791.465,E2 23791.465} C_VEL
LIN {X 0,Y 116.087,Z 762.435,A -85,B 0,C 180,E1 23804.657,E2 23804.657} C_VEL
LIN {X 0,Y 110.927,Z 764.206,A -85,B 0,C 180,E1 23817.03,E2 23817.03} C_VEL
LIN {X 0,Y 110.812,Z 761.014,A -85,B 0,C 180,E1 23832.439,E2 23832.439} C_VEL
LIN {X 0,Y 115.897,Z 752.572,A -85,B 0,C 180,E1 23846.264,E2 23846.264} C_VEL
LIN {X 0,Y 124.514,Z 739.128,A -85,B 0,C 180,E1 23857.833,E2 23857.833} C_VEL
LIN {X 0,Y 127.992,Z 733.711,A -85,B 0,C 180,E1 23861.011,E2 23861.011} C_VEL
LIN {X 0,Y 131.229,Z 723.087,A -85,B 0,C 180,E1 23867.029,E2 23867.029} C_VEL
LIN {X 0,Y 134.149,Z 712.541,A -85,B 0,C 180,E1 23871.693,E2 23871.693} C_VEL
LIN {X 0,Y 134.965,Z 710.874,A -85,B 0,C 180,E1 23872.188,E2 23872.188} C_VEL
LIN {X 0,Y 146.253,Z 686.017,A -85,B 0,C 180,E1 23877.683,E2 23877.683} C_VEL
LIN {X 0,Y 154.806,Z 658.393,A -85,B 0,C 180,E1 23881.135,E2 23881.135} C_VEL
LIN {X 0,Y 156.238,Z 649.909,A -85,B 0,C 180,E1 23881.99,E2 23881.99} C_VEL
LIN {X 0,Y 149.778,Z 653.832,A -85,B 0,C 180,E1 23884.311,E2 23884.311} C_VEL
LIN {X 0,Y 139.066,Z 666.551,A -85,B 0,C 180,E1 23887.079,E2 23887.079} C_VEL
LIN {X 0,Y 131.999,Z 671.18,A -85,B 0,C 180,E1 23890.124,E2 23890.124} C_VEL
LIN {X 0,Y 116.926,Z 703.283,A -85,B 0,C 180,E1 23902.181,E2 23902.181} C_VEL
LIN {X 0,Y 107.492,Z 726.121,A -85,B 0,C 180,E1 23916.199,E2 23916.199} C_VEL
LIN {X 0,Y 103.455,Z 742.529,A -85,B 0,C 180,E1 23931.602,E2 23931.602} C_VEL
LIN {X 0,Y 103.49,Z 753.207,A -85,B 0,C 180,E1 23946.267,E2 23946.267} C_VEL
LIN {X 0,Y 109.854,Z 762.249,A -85,B 0,C 180,E1 23964.324,E2 23964.324} C_VEL
LIN {X 0,Y 127.573,Z 767.956,A -85,B 0,C 180,E1 23980.828,E2 23980.828} C_VEL
LIN {X 0,Y 125.395,Z 768.301,A -85,B 0,C 180,E1 23983.782,E2 23983.782} C_VEL
LIN {X 0,Y 106.848,Z 767.08,A -85,B 0,C 180,E1 24004.936,E2 24004.936} C_VEL
LIN {X 0,Y 104.522,Z 766.367,A -85,B 0,C 180,E1 24011.958,E2 24011.958} C_VEL
LIN {X 0,Y 102.603,Z 772.473,A -85,B 0,C 180,E1 24025.787,E2 24025.787} C_VEL
LIN {X 0,Y 102.845,Z 773.448,A -85,B 0,C 180,E1 24030.004,E2 24030.004} C_VEL
LIN {X 0,Y 102.624,Z 774.139,A -85,B 0,C 180,E1 24038.459,E2 24038.459} C_VEL
LIN {X 0,Y 105.346,Z 772.061,A -85,B 0,C 180,E1 24052.196,E2 24052.196} C_VEL
LIN {X 0,Y 114.572,Z 764.406,A -85,B 0,C 180,E1 24067.25,E2 24067.25} C_VEL
LIN {X 0,Y 128.915,Z 751.443,A -85,B 0,C 180,E1 24078.989,E2 24078.989} C_VEL
LIN {X 0,Y 145.396,Z 733.614,A -85,B 0,C 180,E1 24087.338,E2 24087.338} C_VEL
LIN {X 0,Y 161.646,Z 710.9,A -85,B 0,C 180,E1 24093.216,E2 24093.216} C_VEL
LIN {X 0,Y 175.562,Z 684.021,A -85,B 0,C 180,E1 24097.152,E2 24097.152} C_VEL
LIN {X 0,Y 181.218,Z 668.159,A -85,B 0,C 180,E1 24098.795,E2 24098.795} C_VEL
LIN {X 0,Y 186.468,Z 635.708,A -85,B 0,C 180,E1 24107.776,E2 24107.776} C_VEL
LIN {X 0,Y 187.27,Z 630.627,A -85,B 0,C 180,E1 24109.268,E2 24109.268} C_VEL
LIN {X 0,Y 187.898,Z 631.796,A -85,B 0,C 180,E1 24112.713,E2 24112.713} C_VEL
LIN {X 0,Y 189.486,Z 639.858,A -85,B 0,C 180,E1 24118.152,E2 24118.152} C_VEL
LIN {X 0,Y 190.442,Z 648.686,A -85,B 0,C 180,E1 24121.7,E2 24121.7} C_VEL
LIN {X 0,Y 181.485,Z 678.245,A -85,B 0,C 180,E1 24123.801,E2 24123.801} C_VEL
LIN {X 0,Y 168.932,Z 703.452,A -85,B 0,C 180,E1 24126.974,E2 24126.974} C_VEL
LIN {X 0,Y 153.156,Z 725.629,A -85,B 0,C 180,E1 24131.931,E2 24131.931} C_VEL
LIN {X 0,Y 136.565,Z 742.954,A -85,B 0,C 180,E1 24138.961,E2 24138.961} C_VEL
LIN {X 0,Y 120.86,Z 755.617,A -85,B 0,C 180,E1 24149.069,E2 24149.069} C_VEL
LIN {X 0,Y 110.343,Z 762.226,A -85,B 0,C 180,E1 24160.707,E2 24160.707} C_VEL
LIN {X 0,Y 103.661,Z 764.579,A -85,B 0,C 180,E1 24174.385,E2 24174.385} C_VEL
LIN {X 0,Y 102.296,Z 762.734,A -85,B 0,C 180,E1 24188.356,E2 24188.356} C_VEL
LIN {X 0,Y 106.363,Z 755.846,A -85,B 0,C 180,E1 24203.354,E2 24203.354} C_VEL
LIN {X 0,Y 114.846,Z 743.366,A -85,B 0,C 180,E1 24216.691,E2 24216.691} C_VEL
LIN {X 0,Y 126.58,Z 725.529,A -85,B 0,C 180,E1 24227.008,E2 24227.008} C_VEL
LIN {X 0,Y 134.965,Z 710.874,A -85,B 0,C 180,E1 24232.188,E2 24232.188} C_VEL
LIN {X 0,Y 137.458,Z 704.249,A -85,B 0,C 180,E1 24234.307,E2 24234.307} C_VEL
LIN {X 0,Y 141.459,Z 684.961,A -85,B 0,C 180,E1 24240.152,E2 24240.152} C_VEL
LIN {X 0,Y 142.163,Z 683.029,A -85,B 0,C 180,E1 24240.469,E2 24240.469} C_VEL
LIN {X 0,Y 147.355,Z 667.216,A -85,B 0,C 180,E1 24242.567,E2 24242.567} C_VEL
LIN {X 0,Y 146.662,Z 665.724,A -85,B 0,C 180,E1 24243.271,E2 24243.271} C_VEL
LIN {X 0,Y 135.71,Z 675.544,A -85,B 0,C 180,E1 24246.266,E2 24246.266} C_VEL
LIN {X 0,Y 130.108,Z 679.141,A -85,B 0,C 180,E1 24248.463,E2 24248.463} C_VEL
LIN {X 0,Y 121.114,Z 686.446,A -85,B 0,C 180,E1 24251.607,E2 24251.607} C_VEL
LIN {X 0,Y 115.961,Z 688.994,A -85,B 0,C 180,E1 24254.858,E2 24254.858} C_VEL
LIN {X 0,Y 103.739,Z 715.065,A -85,B 0,C 180,E1 24268.165,E2 24268.165} C_VEL
LIN {X 0,Y 96.638,Z 735.735,A -85,B 0,C 180,E1 24285.289,E2 24285.289} C_VEL
LIN {X 0,Y 95.376,Z 749.208,A -85,B 0,C 180,E1 24302.255,E2 24302.255} C_VEL
LIN {X 0,Y 100.365,Z 759.799,A -85,B 0,C 180,E1 24322.066,E2 24322.066} C_VEL
LIN {X 0,Y 118.168,Z 767.207,A -85,B 0,C 180,E1 24341.053,E2 24341.053} C_VEL
LIN {X 0,Y 115.24,Z 767.362,A -85,B 0,C 180,E1 24344.369,E2 24344.369} C_VEL
LIN {X 0,Y 97.707,Z 764.464,A -85,B 0,C 180,E1 24368.653,E2 24368.653} C_VEL
LIN {X 0,Y 94.733,Z 771.916,A -85,B 0,C 180,E1 24385.436,E2 24385.436} C_VEL
LIN {X 0,Y 94.934,Z 772.938,A -85,B 0,C 180,E1 24390.004,E2 24390.004} C_VEL
LIN {X 0,Y 94.748,Z 773.724,A -85,B 0,C 180,E1 24399.168,E2 24399.168} C_VEL
LIN {X 0,Y 96.856,Z 772.566,A -85,B 0,C 180,E1 24410.842,E2 24410.842} C_VEL
LIN {X 0,Y 106.599,Z 765.69,A -85,B 0,C 180,E1 24428.041,E2 24428.041} C_VEL
LIN {X 0,Y 121.353,Z 753.946,A -85,B 0,C 180,E1 24440.331,E2 24440.331} C_VEL
LIN {X 0,Y 140.038,Z 735.721,A -85,B 0,C 180,E1 24449.553,E2 24449.553} C_VEL
LIN {X 0,Y 157.56,Z 713.517,A -85,B 0,C 180,E1 24455.489,E2 24455.489} C_VEL
LIN {X 0,Y 172.215,Z 687.594,A -85,B 0,C 180,E1 24459.33,E2 24459.33} C_VEL
LIN {X 0,Y 178.919,Z 670.678,A -85,B 0,C 180,E1 24461.232,E2 24461.232} C_VEL
LIN {X 0,Y 186.212,Z 638.725,A -85,B 0,C 180,E1 24470.22,E2 24470.22} C_VEL
LIN {X 0,Y 186.734,Z 640.418,A -85,B 0,C 180,E1 24473.284,E2 24473.284} C_VEL
LIN {X 0,Y 187.584,Z 650.506,A -85,B 0,C 180,E1 24478.862,E2 24478.862} C_VEL
LIN {X 0,Y 187.275,Z 653.918,A -85,B 0,C 180,E1 24479.656,E2 24479.656} C_VEL
LIN {X 0,Y 177.491,Z 682.31,A -85,B 0,C 180,E1 24481.752,E2 24481.752} C_VEL
LIN {X 0,Y 163.463,Z 707.845,A -85,B 0,C 180,E1 24485.128,E2 24485.128} C_VEL
LIN {X 0,Y 146.161,Z 729.86,A -85,B 0,C 180,E1 24490.383,E2 24490.383} C_VEL
LIN {X 0,Y 128.649,Z 746.279,A -85,B 0,C 180,E1 24497.843,E2 24497.843} C_VEL
LIN {X 0,Y 112.837,Z 757.531,A -85,B 0,C 180,E1 24508.258,E2 24508.258} C_VEL
LIN {X 0,Y 101.262,Z 763.642,A -85,B 0,C 180,E1 24521.828,E2 24521.828} C_VEL
LIN {X 0,Y 96.591,Z 764.948,A -85,B 0,C 180,E1 24531.382,E2 24531.382} C_VEL
LIN {X 0,Y 94.272,Z 763.513,A -85,B 0,C 180,E1 24546.407,E2 24546.407} C_VEL
LIN {X 0,Y 98.204,Z 756.804,A -85,B 0,C 180,E1 24563.274,E2 24563.274} C_VEL
LIN {X 0,Y 107.406,Z 744.121,A -85,B 0,C 180,E1 24578.073,E2 24578.073} C_VEL
LIN {X 0,Y 119.98,Z 726.163,A -85,B 0,C 180,E1 24589.012,E2 24589.012} C_VEL
LIN {X 0,Y 133.027,Z 703.435,A -85,B 0,C 180,E1 24596.526,E2 24596.526} C_VEL
LIN {X 0,Y 142.163,Z 683.029,A -85,B 0,C 180,E1 24600.469,E2 24600.469} C_VEL
LIN {X 0,Y 140.807,Z 681.033,A -85,B 0,C 180,E1 24601.773,E2 24601.773} C_VEL
LIN {X 0,Y 134.19,Z 683.142,A -85,B 0,C 180,E1 24604.449,E2 24604.449} C_VEL
LIN {X 0,Y 117.354,Z 693.741,A -85,B 0,C 180,E1 24610.546,E2 24610.546} C_VEL
LIN {X 0,Y 104.881,Z 701.18,A -85,B 0,C 180,E1 24616.875,E2 24616.875} C_VEL
LIN {X 0,Y 101.501,Z 702.828,A -85,B 0,C 180,E1 24620.11,E2 24620.11} C_VEL
LIN {X 0,Y 91.725,Z 724.879,A -85,B 0,C 180,E1 24635.495,E2 24635.495} C_VEL
LIN {X 0,Y 87.736,Z 740.819,A -85,B 0,C 180,E1 24652.575,E2 24652.575} C_VEL
LIN {X 0,Y 88.475,Z 751.92,A -85,B 0,C 180,E1 24669.807,E2 24669.807} C_VEL
LIN {X 0,Y 98.621,Z 762.246,A -85,B 0,C 180,E1 24691.98,E2 24691.98} C_VEL
LIN {X 0,Y 108.172,Z 765.808,A -85,B 0,C 180,E1 24700.849,E2 24700.849} C_VEL
LIN {X 0,Y 107.603,Z 766.053,A -85,B 0,C 180,E1 24703.048,E2 24703.048} C_VEL
LIN {X 0,Y 90.488,Z 763.4,A -85,B 0,C 180,E1 24726.397,E2 24726.397} C_VEL
LIN {X 0,Y 87.135,Z 769.881,A -85,B 0,C 180,E1 24740.032,E2 24740.032} C_VEL
LIN {X 0,Y 87.031,Z 772.426,A -85,B 0,C 180,E1 24750.004,E2 24750.004} C_VEL
LIN {X 0,Y 86.914,Z 773.307,A -85,B 0,C 180,E1 24760.003,E2 24760.003} C_VEL
LIN {X 0,Y 92.163,Z 770.708,A -85,B 0,C 180,E1 24779.424,E2 24779.424} C_VEL
LIN {X 0,Y 105.476,Z 762.322,A -85,B 0,C 180,E1 24795.675,E2 24795.675} C_VEL
LIN {X 0,Y 123.579,Z 748.321,A -85,B 0,C 180,E1 24807.152,E2 24807.152} C_VEL
LIN {X 0,Y 143.304,Z 728.902,A -85,B 0,C 180,E1 24814.85,E2 24814.85} C_VEL
LIN {X 0,Y 160.875,Z 705.433,A -85,B 0,C 180,E1 24819.723,E2 24819.723} C_VEL
LIN {X 0,Y 174.613,Z 679.379,A -85,B 0,C 180,E1 24822.803,E2 24822.803} C_VEL
LIN {X 0,Y 176.615,Z 674.341,A -85,B 0,C 180,E1 24823.405,E2 24823.405} C_VEL
LIN {X 0,Y 184.912,Z 646.673,A -85,B 0,C 180,E1 24831.39,E2 24831.39} C_VEL
LIN {X 0,Y 185.01,Z 654.589,A -85,B 0,C 180,E1 24836.654,E2 24836.654} C_VEL
LIN {X 0,Y 184.708,Z 657.125,A -85,B 0,C 180,E1 24837.435,E2 24837.435} C_VEL
LIN {X 0,Y 174.584,Z 684.537,A -85,B 0,C 180,E1 24839.442,E2 24839.442} C_VEL
LIN {X 0,Y 159.963,Z 709.667,A -85,B 0,C 180,E1 24842.7,E2 24842.7} C_VEL
LIN {X 0,Y 142.891,Z 730.198,A -85,B 0,C 180,E1 24847.472,E2 24847.472} C_VEL
LIN {X 0,Y 124.728,Z 746.398,A -85,B 0,C 180,E1 24854.553,E2 24854.553} C_VEL
LIN {X 0,Y 107.645,Z 757.763,A -85,B 0,C 180,E1 24864.881,E2 24864.881} C_VEL
LIN {X 0,Y 94.065,Z 764.209,A -85,B 0,C 180,E1 24879.933,E2 24879.933} C_VEL
LIN {X 0,Y 86.809,Z 765.023,A -85,B 0,C 180,E1 24898.563,E2 24898.563} C_VEL
LIN {X 0,Y 87.702,Z 761.015,A -85,B 0,C 180,E1 24915.803,E2 24915.803} C_VEL
LIN {X 0,Y 94.593,Z 751.792,A -85,B 0,C 180,E1 24932.282,E2 24932.282} C_VEL
LIN {X 0,Y 105.975,Z 737.213,A -85,B 0,C 180,E1 24945.481,E2 24945.481} C_VEL
LIN {X 0,Y 119.846,Z 716.989,A -85,B 0,C 180,E1 24955.144,E2 24955.144} C_VEL
LIN {X 0,Y 132.711,Z 693.186,A -85,B 0,C 180,E1 24961.214,E2 24961.214} C_VEL
LIN {X 0,Y 137.758,Z 681.221,A -85,B 0,C 180,E1 24963.206,E2 24963.206} C_VEL
LIN {X 0,Y 130.538,Z 684.694,A -85,B 0,C 180,E1 24965.97,E2 24965.97} C_VEL
LIN {X 0,Y 121.107,Z 691.82,A -85,B 0,C 180,E1 24968.84,E2 24968.84} C_VEL
LIN {X 0,Y 117.354,Z 693.741,A -85,B 0,C 180,E1 24970.546,E2 24970.546} C_VEL
LIN {X 0,Y 111.144,Z 698.733,A -85,B 0,C 180,E1 24972.543,E2 24972.543} C_VEL
LIN {X 0,Y 102.192,Z 706.763,A -85,B 0,C 180,E1 24974.785,E2 24974.785} C_VEL
LIN {X 0,Y 100.755,Z 707.498,A -85,B 0,C 180,E1 24975.615,E2 24975.615} C_VEL
LIN {X 0,Y 88.955,Z 713.311,A -85,B 0,C 180,E1 24985.058,E2 24985.058} C_VEL
LIN {X 0,Y 85.897,Z 719.157,A -85,B 0,C 180,E1 24990.621,E2 24990.621} C_VEL
LIN {X 0,Y 80.205,Z 737.796,A -85,B 0,C 180,E1 25010.51,E2 25010.51} C_VEL
LIN {X 0,Y 80.859,Z 750.454,A -85,B 0,C 180,E1 25030.741,E2 25030.741} C_VEL
LIN {X 0,Y 93.717,Z 762.12,A -85,B 0,C 180,E1 25056.389,E2 25056.389} C_VEL
LIN {X 0,Y 98.252,Z 763.886,A -85,B 0,C 180,E1 25060.595,E2 25060.595} C_VEL
LIN {X 0,Y 98.611,Z 764.301,A -85,B 0,C 180,E1 25062.793,E2 25062.793} C_VEL
LIN {X 0,Y 84.217,Z 761.389,A -85,B 0,C 180,E1 25082.336,E2 25082.336} C_VEL
LIN {X 0,Y 79.32,Z 769.23,A -85,B 0,C 180,E1 25099.038,E2 25099.038} C_VEL
LIN {X 0,Y 79.117,Z 771.908,A -85,B 0,C 180,E1 25110.005,E2 25110.005} C_VEL
LIN {X 0,Y 80.935,Z 772.483,A -85,B 0,C 180,E1 25131.256,E2 25131.256} C_VEL
LIN {X 0,Y 91.673,Z 767.204,A -85,B 0,C 180,E1 25151.185,E2 25151.185} C_VEL
LIN {X 0,Y 109.78,Z 755.995,A -85,B 0,C 180,E1 25165.567,E2 25165.567} C_VEL
LIN {X 0,Y 129.683,Z 740.151,A -85,B 0,C 180,E1 25174.4,E2 25174.4} C_VEL
LIN {X 0,Y 150.144,Z 718.333,A -85,B 0,C 180,E1 25180.434,E2 25180.434} C_VEL
LIN {X 0,Y 166.636,Z 693.919,A -85,B 0,C 180,E1 25184.036,E2 25184.036} C_VEL
LIN {X 0,Y 174.539,Z 677.835,A -85,B 0,C 180,E1 25185.654,E2 25185.654} C_VEL
LIN {X 0,Y 182.87,Z 655.722,A -85,B 0,C 180,E1 25192.307,E2 25192.307} C_VEL
LIN {X 0,Y 182.445,Z 660.063,A -85,B 0,C 180,E1 25194.995,E2 25194.995} C_VEL
LIN {X 0,Y 171.46,Z 687.715,A -85,B 0,C 180,E1 25197.138,E2 25197.138} C_VEL
LIN {X 0,Y 156.43,Z 711.872,A -85,B 0,C 180,E1 25200.239,E2 25200.239} C_VEL
LIN {X 0,Y 137.722,Z 732.911,A -85,B 0,C 180,E1 25205.139,E2 25205.139} C_VEL
LIN {X 0,Y 118.288,Z 748.675,A -85,B 0,C 180,E1 25212.426,E2 25212.426} C_VEL
LIN {X 0,Y 99.181,Z 759.869,A -85,B 0,C 180,E1 25224.086,E2 25224.086} C_VEL
LIN {X 0,Y 90.217,Z 763.718,A -85,B 0,C 180,E1 25233.239,E2 25233.239} C_VEL
LIN {X 0,Y 81.754,Z 765.757,A -85,B 0,C 180,E1 25247.607,E2 25247.607} C_VEL
LIN {X 0,Y 78.522,Z 763.801,A -85,B 0,C 180,E1 25267.392,E2 25267.392} C_VEL
LIN {X 0,Y 83.655,Z 756.397,A -85,B 0,C 180,E1 25287.366,E2 25287.366} C_VEL
LIN {X 0,Y 93.883,Z 744.244,A -85,B 0,C 180,E1 25302.734,E2 25302.734} C_VEL
LIN {X 0,Y 107.907,Z 726.47,A -85,B 0,C 180,E1 25314.116,E2 25314.116} C_VEL
LIN {X 0,Y 122.256,Z 703.75,A -85,B 0,C 180,E1 25321.708,E2 25321.708} C_VEL
LIN {X 0,Y 127.686,Z 692.701,A -85,B 0,C 180,E1 25324.167,E2 25324.167} C_VEL
LIN {X 0,Y 115.42,Z 699.918,A -85,B 0,C 180,E1 25328.316,E2 25328.316} C_VEL
LIN {X 0,Y 100.755,Z 707.498,A -85,B 0,C 180,E1 25335.615,E2 25335.615} C_VEL
LIN {X 0,Y 94.546,Z 711.829,A -85,B 0,C 180,E1 25338.404,E2 25338.404} C_VEL
LIN {X 0,Y 85.479,Z 718.75,A -85,B 0,C 180,E1 25342.015,E2 25342.015} C_VEL
LIN {X 0,Y 84.235,Z 719.365,A -85,B 0,C 180,E1 25343.167,E2 25343.167} C_VEL
LIN {X 0,Y 75.806,Z 723.834,A -85,B 0,C 180,E1 25355.199,E2 25355.199} C_VEL
LIN {X 0,Y 72.02,Z 740.536,A -85,B 0,C 180,E1 25376.981,E2 25376.981} C_VEL
LIN {X 0,Y 74.552,Z 751.503,A -85,B 0,C 180,E1 25397.658,E2 25397.658} C_VEL
LIN {X 0,Y 90.241,Z 762.207,A -85,B 0,C 180,E1 25421.962,E2 25421.962} C_VEL
LIN {X 0,Y 78.246,Z 759.428,A -85,B 0,C 180,E1 25437.977,E2 25437.977} C_VEL
LIN {X 0,Y 71.556,Z 768.531,A -85,B 0,C 180,E1 25457.831,E2 25457.831} C_VEL
LIN {X 0,Y 71.201,Z 771.366,A -85,B 0,C 180,E1 25470.005,E2 25470.005} C_VEL
LIN {X 0,Y 71.248,Z 772.469,A -85,B 0,C 180,E1 25482.233,E2 25482.233} C_VEL
LIN {X 0,Y 78.525,Z 770.329,A -85,B 0,C 180,E1 25505.211,E2 25505.211} C_VEL
LIN {X 0,Y 94.901,Z 762.506,A -85,B 0,C 180,E1 25522.665,E2 25522.665} C_VEL
LIN {X 0,Y 115.669,Z 749.367,A -85,B 0,C 180,E1 25533.776,E2 25533.776} C_VEL
LIN {X 0,Y 137.162,Z 731.076,A -85,B 0,C 180,E1 25540.738,E2 25540.738} C_VEL
LIN {X 0,Y 156.213,Z 708.942,A -85,B 0,C 180,E1 25545.022,E2 25545.022} C_VEL
LIN {X 0,Y 172.279,Z 682.08,A -85,B 0,C 180,E1 25547.882,E2 25547.882} C_VEL
LIN {X 0,Y 178.631,Z 668.163,A -85,B 0,C 180,E1 25551.838,E2 25551.838} C_VEL
LIN {X 0,Y 179.441,Z 666.738,A -85,B 0,C 180,E1 25553.009,E2 25553.009} C_VEL
LIN {X 0,Y 167.384,Z 693.163,A -85,B 0,C 180,E1 25554.98,E2 25554.98} C_VEL
LIN {X 0,Y 150.983,Z 716.811,A -85,B 0,C 180,E1 25558.16,E2 25558.16} C_VEL
LIN {X 0,Y 130.539,Z 737.428,A -85,B 0,C 180,E1 25563.277,E2 25563.277} C_VEL
LIN {X 0,Y 109.606,Z 752.337,A -85,B 0,C 180,E1 25571.141,E2 25571.141} C_VEL
LIN {X 0,Y 90.079,Z 762.006,A -85,B 0,C 180,E1 25583.688,E2 25583.688} C_VEL
LIN {X 0,Y 77.585,Z 765.811,A -85,B 0,C 180,E1 25598.916,E2 25598.916} C_VEL
LIN {X 0,Y 70.943,Z 765.509,A -85,B 0,C 180,E1 25618.331,E2 25618.331} C_VEL
LIN {X 0,Y 72.185,Z 761.252,A -85,B 0,C 180,E1 25637.928,E2 25637.928} C_VEL
LIN {X 0,Y 81.187,Z 751.079,A -85,B 0,C 180,E1 25658.009,E2 25658.009} C_VEL
LIN {X 0,Y 95.308,Z 735.271,A -85,B 0,C 180,E1 25672.451,E2 25672.451} C_VEL
LIN {X 0,Y 111.023,Z 714.241,A -85,B 0,C 180,E1 25681.777,E2 25681.777} C_VEL
LIN {X 0,Y 115.94,Z 706.275,A -85,B 0,C 180,E1 25684.051,E2 25684.051} C_VEL
LIN {X 0,Y 115.38,Z 705.054,A -85,B 0,C 180,E1 25685.158,E2 25685.158} C_VEL
LIN {X 0,Y 97.799,Z 713.37,A -85,B 0,C 180,E1 25692.945,E2 25692.945} C_VEL
LIN {X 0,Y 84.235,Z 719.365,A -85,B 0,C 180,E1 25703.167,E2 25703.167} C_VEL
LIN {X 0,Y 78.665,Z 722.981,A -85,B 0,C 180,E1 25707.272,E2 25707.272} C_VEL
LIN {X 0,Y 69.846,Z 729.311,A -85,B 0,C 180,E1 25713.463,E2 25713.463} C_VEL
LIN {X 0,Y 69.166,Z 729.717,A -85,B 0,C 180,E1 25714.501,E2 25714.501} C_VEL
LIN {X 0,Y 64.978,Z 733.146,A -85,B 0,C 180,E1 25728.258,E2 25728.258} C_VEL
LIN {X 0,Y 65.791,Z 746.938,A -85,B 0,C 180,E1 25753.241,E2 25753.241} C_VEL
LIN {X 0,Y 80.424,Z 759.336,A -85,B 0,C 180,E1 25781.707,E2 25781.707} C_VEL
LIN {X 0,Y 72.535,Z 757.578,A -85,B 0,C 180,E1 25793.272,E2 25793.272} C_VEL
LIN {X 0,Y 63.808,Z 767.818,A -85,B 0,C 180,E1 25816.327,E2 25816.327} C_VEL
LIN {X 0,Y 63.285,Z 770.779,A -85,B 0,C 180,E1 25830.006,E2 25830.006} C_VEL
LIN {X 0,Y 64.673,Z 772.075,A -85,B 0,C 180,E1 25851.095,E2 25851.095} C_VEL
LIN {X 0,Y 75.895,Z 768.811,A -85,B 0,C 180,E1 25874.105,E2 25874.105} C_VEL
LIN {X 0,Y 95.749,Z 759.804,A -85,B 0,C 180,E1 25890.096,E2 25890.096} C_VEL
LIN {X 0,Y 118.782,Z 745.351,A -85,B 0,C 180,E1 25899.548,E2 25899.548} C_VEL
LIN {X 0,Y 140.493,Z 726.581,A -85,B 0,C 180,E1 25905.174,E2 25905.174} C_VEL
LIN {X 0,Y 159.932,Z 703.044,A -85,B 0,C 180,E1 25908.707,E2 25908.707} C_VEL
LIN {X 0,Y 171.975,Z 682.967,A -85,B 0,C 180,E1 25910.81,E2 25910.81} C_VEL
LIN {X 0,Y 172.562,Z 681.99,A -85,B 0,C 180,E1 25911.384,E2 25911.384} C_VEL
LIN {X 0,Y 157.388,Z 707.324,A -85,B 0,C 180,E1 25913.714,E2 25913.714} C_VEL
LIN {X 0,Y 137.457,Z 729.899,A -85,B 0,C 180,E1 25917.649,E2 25917.649} C_VEL
LIN {X 0,Y 116.98,Z 746.217,A -85,B 0,C 180,E1 25923.214,E2 25923.214} C_VEL
LIN {X 0,Y 94.769,Z 758.563,A -85,B 0,C 180,E1 25932.85,E2 25932.85} C_VEL
LIN {X 0,Y 75.904,Z 765.254,A -85,B 0,C 180,E1 25948.55,E2 25948.55} C_VEL
LIN {X 0,Y 65.709,Z 766.557,A -85,B 0,C 180,E1 25966.446,E2 25966.446} C_VEL
LIN {X 0,Y 63.204,Z 763.114,A -85,B 0,C 180,E1 25992.805,E2 25992.805} C_VEL
LIN {X 0,Y 69.631,Z 755.882,A -85,B 0,C 180,E1 26013.1,E2 26013.1} C_VEL
LIN {X 0,Y 83.544,Z 741.708,A -85,B 0,C 180,E1 26031.172,E2 26031.172} C_VEL
LIN {X 0,Y 99.943,Z 722.661,A -85,B 0,C 180,E1 26042.162,E2 26042.162} C_VEL
LIN {X 0,Y 105.64,Z 714.881,A -85,B 0,C 180,E1 26044.842,E2 26044.842} C_VEL
LIN {X 0,Y 73.12,Z 727.863,A -85,B 0,C 180,E1 26067.859,E2 26067.859} C_VEL
LIN {X 0,Y 69.166,Z 729.717,A -85,B 0,C 180,E1 26074.501,E2 26074.501} C_VEL
LIN {X 0,Y 61.004,Z 735.977,A -85,B 0,C 180,E1 26087.212,E2 26087.212} C_VEL
LIN {X 0,Y 56.636,Z 741.421,A -85,B 0,C 180,E1 26102.895,E2 26102.895} C_VEL
LIN {X 0,Y 58.39,Z 744.865,A -85,B 0,C 180,E1 26114.956,E2 26114.956} C_VEL
LIN {X 0,Y 69.823,Z 755.479,A -85,B 0,C 180,E1 26140.395,E2 26140.395} C_VEL
LIN {X 0,Y 70.63,Z 756.159,A -85,B 0,C 180,E1 26143.54,E2 26143.54} C_VEL
LIN {X 0,Y 67.445,Z 755.635,A -85,B 0,C 180,E1 26147.847,E2 26147.847} C_VEL
LIN {X 0,Y 57.134,Z 765.665,A -85,B 0,C 180,E1 26169.274,E2 26169.274} C_VEL
LIN {X 0,Y 55.382,Z 770.189,A -85,B 0,C 180,E1 26190.007,E2 26190.007} C_VEL
LIN {X 0,Y 55.754,Z 771.545,A -85,B 0,C 180,E1 26205.71,E2 26205.71} C_VEL
LIN {X 0,Y 65.994,Z 769.956,A -85,B 0,C 180,E1 26233.319,E2 26233.319} C_VEL
LIN {X 0,Y 86.089,Z 762.751,A -85,B 0,C 180,E1 26251.221,E2 26251.221} C_VEL
LIN {X 0,Y 111.229,Z 749.323,A -85,B 0,C 180,E1 26261.753,E2 26261.753} C_VEL
LIN {X 0,Y 134.352,Z 731.755,A -85,B 0,C 180,E1 26267.468,E2 26267.468} C_VEL
LIN {X 0,Y 152.953,Z 712.388,A -85,B 0,C 180,E1 26270.613,E2 26270.613} C_VEL
LIN {X 0,Y 153.801,Z 711.431,A -85,B 0,C 180,E1 26271.253,E2 26271.253} C_VEL
LIN {X 0,Y 134.383,Z 731.874,A -85,B 0,C 180,E1 26274.672,E2 26274.672} C_VEL
LIN {X 0,Y 112.595,Z 748.006,A -85,B 0,C 180,E1 26280.01,E2 26280.01} C_VEL
LIN {X 0,Y 88.496,Z 760.158,A -85,B 0,C 180,E1 26289.831,E2 26289.831} C_VEL
LIN {X 0,Y 67.757,Z 766.203,A -85,B 0,C 180,E1 26307.011,E2 26307.011} C_VEL
LIN {X 0,Y 59.608,Z 767.005,A -85,B 0,C 180,E1 26320.574,E2 26320.574} C_VEL
LIN {X 0,Y 54.76,Z 764.79,A -85,B 0,C 180,E1 26345.578,E2 26345.578} C_VEL
LIN {X 0,Y 60.402,Z 757.92,A -85,B 0,C 180,E1 26371.588,E2 26371.588} C_VEL
LIN {X 0,Y 74.608,Z 744.801,A -85,B 0,C 180,E1 26392.162,E2 26392.162} C_VEL
LIN {X 0,Y 91.129,Z 727.514,A -85,B 0,C 180,E1 26403.775,E2 26403.775} C_VEL
LIN {X 0,Y 93.479,Z 723.655,A -85,B 0,C 180,E1 26406.164,E2 26406.164} C_VEL
LIN {X 0,Y 60.691,Z 736.309,A -85,B 0,C 180,E1 26438.082,E2 26438.082} C_VEL
LIN {X 0,Y 57.183,Z 739.288,A -85,B 0,C 180,E1 26452.398,E2 26452.398} C_VEL
LIN {X 0,Y 56.636,Z 741.421,A -85,B 0,C 180,E1 26462.895,E2 26462.895} C_VEL
LIN {X 0,Y 55.849,Z 745.521,A -85,B 0,C 180,E1 26475.588,E2 26475.588} C_VEL
LIN {X 0,Y 57.033,Z 752.317,A -85,B 0,C 180,E1 26494.68,E2 26494.68} C_VEL
LIN {X 0,Y 57.983,Z 752.815,A -85,B 0,C 180,E1 26496.603,E2 26496.603} C_VEL
LIN {X 0,Y 61.789,Z 754.537,A -85,B 0,C 180,E1 26502.9,E2 26502.9} C_VEL
LIN {X 0,Y 50.108,Z 764.477,A -85,B 0,C 180,E1 26524.56,E2 26524.56} C_VEL
LIN {X 0,Y 47.486,Z 769.588,A -85,B 0,C 180,E1 26550.008,E2 26550.008} C_VEL
LIN {X 0,Y 48.549,Z 771.173,A -85,B 0,C 180,E1 26571.246,E2 26571.246} C_VEL
LIN {X 0,Y 60.393,Z 769.728,A -85,B 0,C 180,E1 26598.563,E2 26598.563} C_VEL
LIN {X 0,Y 82.513,Z 762.885,A -85,B 0,C 180,E1 26616.131,E2 26616.131} C_VEL
LIN {X 0,Y 107.27,Z 750.912,A -85,B 0,C 180,E1 26625.28,E2 26625.28} C_VEL
LIN {X 0,Y 132.655,Z 732.999,A -85,B 0,C 180,E1 26630.737,E2 26630.737} C_VEL
LIN {X 0,Y 132.777,Z 732.913,A -85,B 0,C 180,E1 26631.389,E2 26631.389} C_VEL
LIN {X 0,Y 109.334,Z 749.422,A -85,B 0,C 180,E1 26636.372,E2 26636.372} C_VEL
LIN {X 0,Y 86.781,Z 760.074,A -85,B 0,C 180,E1 26644.233,E2 26644.233} C_VEL
LIN {X 0,Y 64.182,Z 766.387,A -85,B 0,C 180,E1 26659.856,E2 26659.856} C_VEL
LIN {X 0,Y 53.912,Z 767.393,A -85,B 0,C 180,E1 26674.067,E2 26674.067} C_VEL
LIN {X 0,Y 46.938,Z 765.564,A -85,B 0,C 180,E1 26701.16,E2 26701.16} C_VEL
LIN {X 0,Y 52.289,Z 758.798,A -85,B 0,C 180,E1 26732.722,E2 26732.722} C_VEL
LIN {X 0,Y 67.256,Z 746.283,A -85,B 0,C 180,E1 26755.004,E2 26755.004} C_VEL
LIN {X 0,Y 82.157,Z 732.208,A -85,B 0,C 180,E1 26765.684,E2 26765.684} C_VEL
LIN {X 0,Y 79.922,Z 732.32,A -85,B 0,C 180,E1 26767.759,E2 26767.759} C_VEL
LIN {X 0,Y 50.661,Z 743.772,A -85,B 0,C 180,E1 26811.412,E2 26811.412} C_VEL
LIN {X 0,Y 51.336,Z 748.421,A -85,B 0,C 180,E1 26837.071,E2 26837.071} C_VEL
LIN {X 0,Y 57.983,Z 752.815,A -85,B 0,C 180,E1 26856.603,E2 26856.603} C_VEL
LIN {X 0,Y 57.134,Z 755.201,A -85,B 0,C 180,E1 26861.573,E2 26861.573} C_VEL
LIN {X 0,Y 44.449,Z 762.4,A -85,B 0,C 180,E1 26875.801,E2 26875.801} C_VEL
LIN {X 0,Y 39.575,Z 768.971,A -85,B 0,C 180,E1 26910.009,E2 26910.009} C_VEL
LIN {X 0,Y 40.608,Z 770.564,A -85,B 0,C 180,E1 26931.824,E2 26931.824} C_VEL
LIN {X 0,Y 55.385,Z 769.504,A -85,B 0,C 180,E1 26964.834,E2 26964.834} C_VEL
LIN {X 0,Y 79.59,Z 762.988,A -85,B 0,C 180,E1 26981.452,E2 26981.452} C_VEL
LIN {X 0,Y 107.317,Z 750.427,A -85,B 0,C 180,E1 26989.844,E2 26989.844} C_VEL
LIN {X 0,Y 112.254,Z 747.56,A -85,B 0,C 180,E1 26991.291,E2 26991.291} C_VEL
LIN {X 0,Y 85.969,Z 760.017,A -85,B 0,C 180,E1 26998.461,E2 26998.461} C_VEL
LIN {X 0,Y 61.695,Z 766.519,A -85,B 0,C 180,E1 27011.913,E2 27011.913} C_VEL
LIN {X 0,Y 49.885,Z 767.771,A -85,B 0,C 180,E1 27024.823,E2 27024.823} C_VEL
LIN {X 0,Y 40.562,Z 766.898,A -85,B 0,C 180,E1 27048.119,E2 27048.119} C_VEL
LIN {X 0,Y 42.747,Z 760.742,A -85,B 0,C 180,E1 27089.991,E2 27089.991} C_VEL
LIN {X 0,Y 57.093,Z 749.979,A -85,B 0,C 180,E1 27115.584,E2 27115.584} C_VEL
LIN {X 0,Y 69.903,Z 739.514,A -85,B 0,C 180,E1 27126.011,E2 27126.011} C_VEL
LIN {X 0,Y 69.436,Z 738.821,A -85,B 0,C 180,E1 27127.995,E2 27127.995} C_VEL
LIN {X 0,Y 43.104,Z 749.244,A -85,B 0,C 180,E1 27179.973,E2 27179.973} C_VEL
LIN {X 0,Y 52.01,Z 756.263,A -85,B 0,C 180,E1 27220.738,E2 27220.738} C_VEL
LIN {X 0,Y 44.449,Z 762.4,A -85,B 0,C 180,E1 27235.801,E2 27235.801} C_VEL
LIN {X 0,Y 37.946,Z 766.081,A -85,B 0,C 180,E1 27250.958,E2 27250.958} C_VEL
LIN {X 0,Y 31.856,Z 769.455,A -85,B 0,C 180,E1 27286.59,E2 27286.59} C_VEL
LIN {X 0,Y 40.468,Z 770.362,A -85,B 0,C 180,E1 27318.239,E2 27318.239} C_VEL
LIN {X 0,Y 63.778,Z 766.889,A -85,B 0,C 180,E1 27341.174,E2 27341.174} C_VEL
LIN {X 0,Y 90.758,Z 758.185,A -85,B 0,C 180,E1 27351.4,E2 27351.4} C_VEL
LIN {X 0,Y 66.573,Z 765.486,A -85,B 0,C 180,E1 27360.017,E2 27360.017} C_VEL
LIN {X 0,Y 42.214,Z 768.217,A -85,B 0,C 180,E1 27380.973,E2 27380.973} C_VEL
LIN {X 0,Y 31.104,Z 765.702,A -85,B 0,C 180,E1 27420.965,E2 27420.965} C_VEL
LIN {X 0,Y 39.965,Z 757.917,A -85,B 0,C 180,E1 27465.62,E2 27465.62} C_VEL
LIN {X 0,Y 57.808,Z 745.707,A -85,B 0,C 180,E1 27486.724,E2 27486.724} C_VEL
LIN {X 0,Y 57.845,Z 745.079,A -85,B 0,C 180,E1 27488.47,E2 27488.47} C_VEL
LIN {X 0,Y 36.084,Z 752.919,A -85,B 0,C 180,E1 27539.968,E2 27539.968} C_VEL
LIN {X 0,Y 42.367,Z 758.077,A -85,B 0,C 180,E1 27578.671,E2 27578.671} C_VEL
LIN {X 0,Y 38.927,Z 760.984,A -85,B 0,C 180,E1 27587.303,E2 27587.303} C_VEL
LIN {X 0,Y 31.669,Z 768.34,A -85,B 0,C 180,E1 27630.012,E2 27630.012} C_VEL
LIN {X 0,Y 31.856,Z 769.455,A -85,B 0,C 180,E1 27646.59,E2 27646.59} C_VEL
LIN {X 0,Y 33.729,Z 770.221,A -85,B 0,C 180,E1 27669.362,E2 27669.362} C_VEL
LIN {X 0,Y 43.627,Z 769.502,A -85,B 0,C 180,E1 27697.31,E2 27697.31} C_VEL
LIN {X 0,Y 44.531,Z 769.312,A -85,B 0,C 180,E1 27698.138,E2 27698.138} C_VEL
LIN {X 0,Y 69.408,Z 765.019,A -85,B 0,C 180,E1 27711.501,E2 27711.501} C_VEL
LIN {X 0,Y 45.379,Z 768.437,A -85,B 0,C 180,E1 27723.867,E2 27723.867} C_VEL
LIN {X 0,Y 26.584,Z 767.519,A -85,B 0,C 180,E1 27754.638,E2 27754.638} C_VEL
LIN {X 0,Y 28.76,Z 760.853,A -85,B 0,C 180,E1 27821.937,E2 27821.937} C_VEL
LIN {X 0,Y 45.78,Z 750.953,A -85,B 0,C 180,E1 27848.01,E2 27848.01} C_VEL
LIN {X 0,Y 42.146,Z 751.348,A -85,B 0,C 180,E1 27854.23,E2 27854.23} C_VEL
LIN {X 0,Y 29.362,Z 757.525,A -85,B 0,C 180,E1 27914.849,E2 27914.849} C_VEL
LIN {X 0,Y 33.24,Z 760.174,A -85,B 0,C 180,E1 27938.535,E2 27938.535} C_VEL
LIN {X 0,Y 23.766,Z 767.656,A -85,B 0,C 180,E1 27990.016,E2 27990.016} C_VEL
LIN {X 0,Y 35.611,Z 769.978,A -85,B 0,C 180,E1 28047.96,E2 28047.96} C_VEL
LIN {X 0,Y 44.531,Z 769.312,A -85,B 0,C 180,E1 28058.138,E2 28058.138} C_VEL
LIN {X 0,Y 44.412,Z 769.211,A -85,B 0,C 180,E1 28062.959,E2 28062.959} C_VEL
LIN {X 0,Y 37.895,Z 769.163,A -85,B 0,C 180,E1 28072.146,E2 28072.146} C_VEL
LIN {X 0,Y 23.611,Z 768.311,A -85,B 0,C 180,E1 28093.334,E2 28093.334} C_VEL
LIN {X 0,Y 19.571,Z 767.486,A -85,B 0,C 180,E1 28105.185,E2 28105.185} C_VEL
LIN {X 0,Y 20.135,Z 761.98,A -85,B 0,C 180,E1 28186.119,E2 28186.119} C_VEL
LIN {X 0,Y 33.143,Z 755.795,A -85,B 0,C 180,E1 28209.845,E2 28209.845} C_VEL
LIN {X 0,Y 26.972,Z 756.828,A -85,B 0,C 180,E1 28225.93,E2 28225.93} C_VEL
LIN {X 0,Y 23.629,Z 761.212,A -85,B 0,C 180,E1 28291.474,E2 28291.474} C_VEL
LIN {X 0,Y 20.799,Z 763.08,A -85,B 0,C 180,E1 28303.515,E2 28303.515} C_VEL
LIN {X 0,Y 15.847,Z 766.935,A -85,B 0,C 180,E1 28350.023,E2 28350.023} C_VEL
LIN {X 0,Y 32.071,Z 769.546,A -85,B 0,C 180,E1 28420.259,E2 28420.259} C_VEL
LIN {X 0,Y 45.926,Z 768.797,A -85,B 0,C 180,E1 28430.347,E2 28430.347} C_VEL
LIN {X 0,Y 45.666,Z 768.738,A -85,B 0,C 180,E1 28432.508,E2 28432.508} C_VEL
LIN {X 0,Y 30.256,Z 768.854,A -85,B 0,C 180,E1 28443.885,E2 28443.885} C_VEL
LIN {X 0,Y 19.571,Z 767.486,A -85,B 0,C 180,E1 28465.185,E2 28465.185} C_VEL
LIN {X 0,Y 11.418,Z 765.81,A -85,B 0,C 180,E1 28497.736,E2 28497.736} C_VEL
LIN {X 0,Y 11.952,Z 763.018,A -85,B 0,C 180,E1 28557.072,E2 28557.072} C_VEL
LIN {X 0,Y 20.02,Z 759.999,A -85,B 0,C 180,E1 28574.261,E2 28574.261} C_VEL
LIN {X 0,Y 13.973,Z 761.799,A -85,B 0,C 180,E1 28619.917,E2 28619.917} C_VEL
LIN {X 0,Y 14.518,Z 762.513,A -85,B 0,C 180,E1 28640.971,E2 28640.971} C_VEL
LIN {X 0,Y 11.674,Z 763.962,A -85,B 0,C 180,E1 28657.604,E2 28657.604} C_VEL
LIN {X 0,Y 7.918,Z 766.216,A -85,B 0,C 180,E1 28710.047,E2 28710.047} C_VEL
LIN {X 0,Y 16.132,Z 768.373,A -85,B 0,C 180,E1 28779.357,E2 28779.357} C_VEL
LIN {X 0,Y 22.582,Z 768.81,A -85,B 0,C 180,E1 28792.792,E2 28792.792} C_VEL
LIN {X 0,Y 10.589,Z 763.564,A -85,B 0,C 180,E1 28910.834,E2 28910.834} C_VEL
LIN {X 0,Y 11.952,Z 763.018,A -85,B 0,C 180,E1 28917.072,E2 28917.072} C_VEL
LIN {X 0,Y 14.046,Z 764.934,A -85,B 0,C 180,E1 28923.675,E2 28923.675} C_VEL
LIN {X 0,Y 14.046,Z 799,A -85,B 0,C 180,E1 28923.675,E2 28923.675} C_VEL
LIN {X 0,Y 14.046,Z 799,A -85,B 0,C 180,E1 28923.675,E2 28923.675}

